(* IEC 61131-3 sources: RL_MAR/experiments/results/ablation/Ablation_antlr_only_deepseek-ai_DeepSeek-V3.2_20260611_164353, 94 files *)

(* ---- hard_92.st ---- *)
FUNCTION_BLOCK FB_BreakerControlSystem
VAR_INPUT
    B10_1_Trip : BOOL;
    B10_1_Close : BOOL;
    B10_2_Trip : BOOL;
    B10_2_Close : BOOL;
    B10_12_Trip : BOOL;
    B10_12_Close : BOOL;
    B54_Trip : BOOL;
    B54_Close : BOOL;
    B55_Trip : BOOL;
    B55_Close : BOOL;
    B56_Trip : BOOL;
    B56_Close : BOOL;
    B57_Trip : BOOL;
    B57_Close : BOOL;
END_VAR

VAR_OUTPUT
    Point_1a : INT;
    Point_2a : INT;
    Point_3a : INT;
    Point_4a : INT;
    B10_1_Opened : BOOL;
    B10_1_Closed : BOOL;
    B10_2_Opened : BOOL;
    B10_2_Closed : BOOL;
    B10_12_Opened : BOOL;
    B10_12_Closed : BOOL;
    B54_Opened : BOOL;
    B54_Closed : BOOL;
    B55_Opened : BOOL;
    B55_Closed : BOOL;
    B56_Opened : BOOL;
    B56_Closed : BOOL;
    B57_Opened : BOOL;
    B57_Closed : BOOL;
END_VAR

VAR
    b10_1_state : BOOL := FALSE;
    b10_2_state : BOOL := FALSE;
    b10_12_state : BOOL := FALSE;
    b54_state : BOOL := FALSE;
    b55_state : BOOL := FALSE;
    b56_state : BOOL := FALSE;
    b57_state : BOOL := FALSE;
END_VAR

(* Breaker B10_1 State Management *)
IF B10_1_Trip THEN
    b10_1_state := FALSE;
ELSIF B10_1_Close THEN
    b10_1_state := TRUE;
END_IF;

B10_1_Closed := b10_1_state;
B10_1_Opened := NOT b10_1_state;

(* Breaker B10_2 State Management *)
IF B10_2_Trip THEN
    b10_2_state := FALSE;
ELSIF B10_2_Close THEN
    b10_2_state := TRUE;
END_IF;

B10_2_Closed := b10_2_state;
B10_2_Opened := NOT b10_2_state;

(* Breaker B10_12 State Management *)
IF B10_12_Trip THEN
    b10_12_state := FALSE;
ELSIF B10_12_Close THEN
    b10_12_state := TRUE;
END_IF;

B10_12_Closed := b10_12_state;
B10_12_Opened := NOT b10_12_state;

(* Breaker B54 State Management *)
IF B54_Trip THEN
    b54_state := FALSE;
ELSIF B54_Close THEN
    b54_state := TRUE;
END_IF;

B54_Closed := b54_state;
B54_Opened := NOT b54_state;

(* Breaker B55 State Management *)
IF B55_Trip THEN
    b55_state := FALSE;
ELSIF B55_Close THEN
    b55_state := TRUE;
END_IF;

B55_Closed := b55_state;
B55_Opened := NOT b55_state;

(* Breaker B56 State Management *)
IF B56_Trip THEN
    b56_state := FALSE;
ELSIF B56_Close THEN
    b56_state := TRUE;
END_IF;

B56_Closed := b56_state;
B56_Opened := NOT b56_state;

(* Breaker B57 State Management *)
IF B57_Trip THEN
    b57_state := FALSE;
ELSIF B57_Close THEN
    b57_state := TRUE;
END_IF;

B57_Closed := b57_state;
B57_Opened := NOT b57_state;

(* Point Calculations *)
(* Point_1a: B54 closed AND ((B10_12 closed AND B10_1 closed) OR B10_2 closed) *)
IF b54_state AND ((b10_12_state AND b10_1_state) OR b10_2_state) THEN
    Point_1a := 0;
ELSE
    Point_1a := 138;
END_IF;

(* Point_2a: B55 closed AND ((B10_12 closed AND B10_1 closed) OR B10_2 closed) *)
IF b55_state AND ((b10_12_state AND b10_1_state) OR b10_2_state) THEN
    Point_2a := 0;
ELSE
    Point_2a := 138;
END_IF;

(* Point_3a: B56 closed AND ((B10_12 closed AND B10_2 closed) OR B10_1 closed) *)
IF b56_state AND ((b10_12_state AND b10_2_state) OR b10_1_state) THEN
    Point_3a := 0;
ELSE
    Point_3a := 138;
END_IF;

(* Point_4a: B57 closed AND ((B10_12 closed AND B10_2 closed) OR B10_1 closed) *)
IF b57_state AND ((b10_12_state AND b10_2_state) OR b10_1_state) THEN
    Point_4a := 0;
ELSE
    Point_4a := 138;
END_IF;

END_FUNCTION_BLOCK;

(* ---- hard_93.st ---- *)
TYPE ST_CircuitBreakerStates :
STRUCT
    Open_CB2_22KV : BOOL;
    Open_CB1_66KV : BOOL;
    Open_CB_TRSF1 : BOOL;
    Open_CB2_66KV : BOOL;
END_STRUCT
END_TYPE

FUNCTION_BLOCK FB_CircuitControl
VAR_INPUT
    Reset_All_CB : BOOL;
    Current_Fault_on_TRSF1 : INT;
    Current_Fault_on_66BUS1 : INT;
END_VAR

VAR_OUTPUT
    Short_Circuit_TRSF1 : BOOL;
    Short_Circuit_66BUS : BOOL;
    Open_CB1_66KV : BOOL;
    Open_CB2_66KV : BOOL;
    Open_CB_TRSF1 : BOOL;
    Open_CB2_22KV : BOOL;
END_VAR

VAR
    Threshold500 : INT := 500;
    Prev_States : ST_CircuitBreakerStates;
    Next_States : ST_CircuitBreakerStates;
    bShortCircuitDetected : BOOL;
END_VAR

(* 1. SHORT CIRCUIT DETECTION (Independent of Reset) *)
Short_Circuit_66BUS := (Current_Fault_on_66BUS1 > Threshold500);
Short_Circuit_TRSF1 := (Current_Fault_on_TRSF1 > Threshold500);

(* 2. RESET OVERRIDE - All breakers to FALSE (Closed) except CB2_66KV *)
IF Reset_All_CB THEN
    Next_States.Open_CB2_22KV := FALSE;
    Next_States.Open_CB1_66KV := FALSE;
    Next_States.Open_CB_TRSF1 := FALSE;
    Next_States.Open_CB2_66KV := TRUE; (* Per specification *)
ELSE
    (* 3. CALCULATE NEXT STATES BASED ON PREVIOUS SCAN CYCLE *)
    (* Initialize with previous state - prevents rapid switching *)
    Next_States := Prev_States;

    (* Combined short circuit flag for logic simplification *)
    bShortCircuitDetected := Short_Circuit_66BUS OR Short_Circuit_TRSF1;

    (* --- FIRST PASS LOGIC (as per specification order) --- *)
    (* Open_CB2_22KV - First Condition *)
    IF (NOT Prev_States.Open_CB2_22KV) AND
       ((Prev_States.Open_CB1_66KV AND Prev_States.Open_CB_TRSF1) OR Short_Circuit_66BUS) THEN
        Next_States.Open_CB2_22KV := TRUE;
    END_IF;

    (* Open_CB1_66KV - First Condition *)
    IF (NOT Next_States.Open_CB2_22KV) AND
       ((Prev_States.Open_CB1_66KV AND Prev_States.Open_CB_TRSF1) OR Short_Circuit_66BUS) THEN
        Next_States.Open_CB1_66KV := TRUE;
    END_IF;

    (* Open_CB_TRSF1 - First Condition *)
    IF (NOT Next_States.Open_CB2_22KV) AND
       ((Next_States.Open_CB1_66KV AND Prev_States.Open_CB_TRSF1) OR Short_Circuit_66BUS) THEN
        Next_States.Open_CB_TRSF1 := TRUE;
    END_IF;

    (* Open_CB2_66KV - Always TRUE per specification *)
    Next_States.Open_CB2_66KV := TRUE;

    (* --- SECOND PASS LOGIC (Updates as per specification) --- *)
    (* Update Open_CB2_22KV again *)
    IF (NOT Prev_States.Open_CB2_22KV) AND
       ((Next_States.Open_CB2_66KV AND Next_States.Open_CB1_66KV AND Next_States.Open_CB_TRSF1) OR Short_Circuit_TRSF1) THEN
        Next_States.Open_CB2_22KV := TRUE;
    END_IF;

    (* Update Open_CB1_66KV again *)
    IF (NOT Next_States.Open_CB2_22KV) AND
       ((Next_States.Open_CB2_66KV AND Prev_States.Open_CB1_66KV AND Next_States.Open_CB_TRSF1) OR Short_Circuit_TRSF1) THEN
        Next_States.Open_CB1_66KV := TRUE;
    END_IF;

    (* Update Open_CB_TRSF1 again *)
    IF (NOT Next_States.Open_CB2_22KV) AND
       ((Next_States.Open_CB2_66KV AND Next_States.Open_CB1_66KV AND Prev_States.Open_CB_TRSF1) OR Short_Circuit_TRSF1) THEN
        Next_States.Open_CB_TRSF1 := TRUE;
    END_IF;

    (* 4. FAILSAFE: If any short circuit is detected, ensure critical breakers open *)
    IF bShortCircuitDetected THEN
        Next_States.Open_CB1_66KV := TRUE;
        Next_States.Open_CB_TRSF1 := TRUE;
        Next_States.Open_CB2_22KV := TRUE;
    END_IF;
END_IF;

(* 5. ASSIGN NEXT STATES TO OUTPUTS *)
Open_CB2_22KV := Next_States.Open_CB2_22KV;
Open_CB1_66KV := Next_States.Open_CB1_66KV;
Open_CB_TRSF1 := Next_States.Open_CB_TRSF1;
Open_CB2_66KV := Next_States.Open_CB2_66KV;

(* 6. STORE CURRENT STATES FOR NEXT SCAN CYCLE *)
Prev_States := Next_States;

END_FUNCTION_BLOCK;

(* ---- hard_94.st ---- *)
FUNCTION_BLOCK FB_AdvancedCircuitBreakerControl
VAR_INPUT
    S_AL1_P_B1 : BOOL;
    S_AL1_P_B2 : BOOL;
    S_AL1_MCB : BOOL;
    MCB_BUSY : BOOL;
    MCB_ERROR : BOOL;
    S_AL1_MCBR : BOOL;
    MCBR_BUSY : BOOL;
    MCBR_ERROR : BOOL;
    S_AL1_P_B3 : BOOL;
    S_AL1_MCB2 : BOOL;
    S_AL1_MCBR2 : BOOL;
END_VAR
VAR_OUTPUT
    E_AL1_B1 : BOOL;
    PUWS_AL1_B1_PLUS : BOOL;
    PUWS_AL1_B1_RIGHT : BOOL;
    PAS_AL1_PLUS : BOOL;
    PAS_AL1_TURN : BOOL;
END_VAR
VAR
    PPAL1 : BOOL := 1;
    PP0 : BOOL := 1;
    PP1 : BOOL := 0;
    PP2 : BOOL := 0;
    PP3 : BOOL := 0;
    PP4 : BOOL := 0;
    MCB : BOOL := 1;
    PP5 : BOOL := 0;
    PP7 : BOOL := 0;
    PPL3 : BOOL := 0;
    PPL4 : BOOL := 0;
    MCBR : BOOL := 1;
    PPL5 : BOOL := 0;
    PPL7 : BOOL := 0;
    STABLE : BOOL := 0;
    MCB_CONTROL : BOOL;
END_VAR

(* State Transition Logic *)
STABLE := 0;
WHILE (STABLE = 0) DO
    STABLE := 1;

    (* Main Path Transitions *)
    IF (PP0 = 1) AND (NOT MCB_CONTROL) AND (PP1 = 0) THEN
        PP0 := 0;
        PP1 := 1;
        STABLE := 0;
    END_IF;

    IF (PP1 = 1) AND S_AL1_P_B1 AND (PP2 = 0) THEN
        PP1 := 0;
        PP2 := 1;
        STABLE := 0;
    END_IF;

    IF (PP2 = 1) AND S_AL1_P_B2 AND (NOT MCB_CONTROL) AND (PP3 = 0) THEN
        PP2 := 0;
        PP3 := 1;
        STABLE := 0;
    END_IF;

    IF (PP3 = 1) AND S_AL1_MCB AND (PP4 = 0) AND (PP1 = 0) THEN
        PP3 := 0;
        PP4 := 1;
        PP1 := 1;
        STABLE := 0;
    END_IF;

    IF (PP4 = 1) AND (MCB = 1) AND MCB_BUSY AND (PP5 = 0) THEN
        PP4 := 0;
        MCB := 0;
        PP5 := 1;
        STABLE := 0;
    END_IF;

    IF (PP5 = 1) AND S_AL1_MCB2 AND (PP7 = 0) AND (MCB = 0) THEN
        PP5 := 0;
        PP7 := 1;
        MCB := 1;
        STABLE := 0;
    END_IF;

    IF (PP7 = 1) AND S_AL1_P_B3 THEN
        PP7 := 0;
        STABLE := 0;
    END_IF;

    (* Alternative Path Transitions *)
    IF (PP2 = 1) AND S_AL1_P_B2 AND MCB_CONTROL AND (PPL3 = 0) AND (PP1 = 0) THEN
        PP2 := 0;
        PPL3 := 1;
        PP1 := 1;
        STABLE := 0;
    END_IF;

    IF (PPL3 = 1) AND S_AL1_MCBR AND (PPL4 = 0) THEN
        PPL3 := 0;
        PPL4 := 1;
        STABLE := 0;
    END_IF;

    IF (PPL4 = 1) AND (MCBR = 1) AND MCBR_BUSY AND (PPL5 = 0) THEN
        PPL4 := 0;
        MCBR := 0;
        PPL5 := 1;
        STABLE := 0;
    END_IF;

    IF (PPL5 = 1) AND S_AL1_MCBR2 AND (PPL7 = 0) AND (MCBR = 0) THEN
        PPL5 := 0;
        PPL7 := 1;
        MCBR := 1;
        STABLE := 0;
    END_IF;

    IF (PPL7 = 1) AND S_AL1_P_B3 THEN
        PPL7 := 0;
        STABLE := 0;
    END_IF;
END_WHILE;

(* Output Control Logic *)
(* E_AL1_B1 - Circuit Activation *)
IF (PP0 = 1) OR (PP1 = 1) THEN
    E_AL1_B1 := 1;
ELSIF (PP2 = 1) OR (PP3 = 1) OR (PPL3 = 1) THEN
    E_AL1_B1 := 0;
ELSE
    E_AL1_B1 := 0;
END_IF;

(* MCB_CONTROL - Main Circuit Breaker Control *)
IF (PP3 = 1) THEN
    MCB_CONTROL := 1;
ELSIF (PP0 = 1) THEN
    MCB_CONTROL := 0;
END_IF;

(* PAS_AL1_PLUS and PAS_AL1_TURN - Process Activation Signals *)
IF (PPL3 = 1) OR (PPL4 = 1) THEN
    PAS_AL1_PLUS := 1;
    PAS_AL1_TURN := 1;
ELSIF (PP0 = 1) OR (PP3 = 1) OR (PP4 = 1) THEN
    PAS_AL1_PLUS := 0;
    PAS_AL1_TURN := 0;
ELSE
    PAS_AL1_PLUS := 0;
    PAS_AL1_TURN := 0;
END_IF;

(* PUWS_AL1_B1_PLUS - Plus Direction Control *)
IF (PPAL1 = 1) OR (PP2 = 1) THEN
    PUWS_AL1_B1_PLUS := 1;
ELSE
    PUWS_AL1_B1_PLUS := 0;
END_IF;

(* PUWS_AL1_B1_RIGHT - Right Direction Control *)
IF (PPAL1 = 1) OR (PP2 = 1) THEN
    PUWS_AL1_B1_RIGHT := 0;
ELSE
    PUWS_AL1_B1_RIGHT := 0;
END_IF;

END_FUNCTION_BLOCK;

(* ---- hf_1.st ---- *)
FUNCTION_BLOCK StackMin
VAR_INPUT
    push : BOOL;
    pop : BOOL;
    reset : BOOL;
END_VAR
VAR_OUTPUT
    error : BOOL;
    status : WORD;
END_VAR
VAR_IN_OUT
    item : INT;
    stack : ARRAY[0..3] OF INT;
END_VAR
VAR
    top : INT := -1; // Tracks the index of the top element; -1 means empty
    i : INT; // Loop counter
    minIndex : INT; // Index of the minimum value found during pop
    minValue : INT; // Minimum value found during pop
END_VAR

// Reset has highest priority
IF reset THEN
    top := -1;
    error := FALSE;
    status := 16#0000;
ELSIF push THEN
    // Check if stack is full
    IF top >= 3 THEN
        error := TRUE;
        status := 16#8A04;
    ELSE
        // Perform push operation
        top := top + 1;
        stack[top] := item;
        error := FALSE;
        status := 16#0000;
    END_IF;
ELSIF pop THEN
    // Check if stack is empty
    IF top < 0 THEN
        error := TRUE;
        status := 16#8A05;
    ELSE
        // Find minimum value and its index
        minIndex := 0;
        minValue := stack[0];

        i := 1;
        WHILE i <= top DO
            IF stack[i] < minValue THEN
                minValue := stack[i];
                minIndex := i;
            END_IF;
            i := i + 1;
        END_WHILE;

        // Return minimum value via item
        item := minValue;

        // Shift elements down to remove the minimum
        i := minIndex;
        WHILE i < top DO
            stack[i] := stack[i + 1];
            i := i + 1;
        END_WHILE;

        // Decrement top
        top := top - 1;

        error := FALSE;
        status := 16#0000;
    END_IF;
ELSE
    // No operation requested
    error := FALSE;
    status := 16#0000;
END_IF;

END_FUNCTION_BLOCK

(* ---- hf_10.st ---- *)
FUNCTION_BLOCK FloatingAverage
VAR_INPUT
    cyclicExecution : BOOL; (* When TRUE, periodic reading is performed, and trigger has no effect *)
    trigger : BOOL; (* External trigger signal, reads value upon each rising edge *)
    value : REAL; (* Newly read data value *)
    windowSize : INT; (* The window size for the moving average, which must be between 1 and 100 *)
    reset : BOOL; (* Reset signal, resets the moving average calculation when TRUE *)
END_VAR
VAR_OUTPUT
    average : REAL; (* The moving average *)
    windowSizeReached : BOOL; (* FALSE: Maximum window width not yet reached, TRUE: Maximum window width has been reached *)
    error : BOOL; (* FALSE: No error occurred, TRUE: An error occurred during the execution of FB *)
    status : WORD; (* Status code *)
END_VAR
VAR
    (* Data buffer and management *)
    dataBuffer : ARRAY[1..100] OF REAL; (* Circular buffer for data values *)
    bufferIndex : INT := 1; (* Current insertion index in the circular buffer *)
    sampleCount : INT := 0; (* Number of valid samples currently in the buffer *)
    sum : REAL := 0.0; (* Running sum of the valid samples in the buffer *)

    (* Edge detection and state tracking *)
    triggerPrev : BOOL := FALSE; (* Previous state of trigger for rising edge detection *)
    cyclicPrev : BOOL := FALSE; (* Previous state of cyclicExecution for edge detection *)

    (* Internal validated window size *)
    internalWindowSize : INT := 1;
END_VAR

(* ================================ *)
(* RESET LOGIC - Highest Priority   *)
(* ================================ *)
IF reset THEN
    (* Clear the data buffer *)
    FOR bufferIndex := 1 TO 100 DO
        dataBuffer[bufferIndex] := 0.0;
    END_FOR;

    (* Reset all internal state variables *)
    bufferIndex := 1;
    sampleCount := 0;
    sum := 0.0;
    triggerPrev := FALSE;
    cyclicPrev := FALSE;

    (* Reset outputs *)
    average := 0.0;
    windowSizeReached := FALSE;
    error := FALSE;
    status := 16#0000; (* Execution successful *)

    (* Validate and set internal window size after reset *)
    IF (windowSize >= 1) AND (windowSize <= 100) THEN
        internalWindowSize := windowSize;
    ELSE
        internalWindowSize := 1; (* Default to minimum valid size *)
    END_IF;

    RETURN; (* Exit function block after reset *)
END_IF;

(* ================================ *)
(* WINDOW SIZE VALIDATION           *)
(* ================================ *)
IF (windowSize < 1) OR (windowSize > 100) THEN
    error := TRUE;
    status := 16#8200; (* Window length setting error *)
    average := 0.0;
    windowSizeReached := FALSE;
    RETURN; (* Exit function block on error *)
ELSE
    error := FALSE;
    status := 16#0000; (* Execution successful *)
    internalWindowSize := windowSize;
END_IF;

(* ================================ *)
(* DATA ACQUISITION LOGIC           *)
(* ================================ *)
IF cyclicExecution THEN
    (* Cyclic mode: process every scan *)
    IF NOT cyclicPrev THEN
        cyclicPrev := TRUE; (* Set for next scan *)

        (* Store the old value that will be overwritten *)
        oldValue : REAL;
        IF sampleCount >= internalWindowSize THEN
            (* Buffer is full, calculate index of oldest value to be overwritten *)
            oldValue := dataBuffer[((bufferIndex - internalWindowSize - 1 + 100) MOD 100) + 1];
        ELSE
            oldValue := 0.0; (* No value to remove when buffer not full *)
        END_IF;

        (* Update buffer with new value *)
        dataBuffer[bufferIndex] := value;

        (* Update running sum *)
        sum := sum + value - oldValue;

        (* Update buffer index (circular) *)
        bufferIndex := (bufferIndex MOD 100) + 1;

        (* Update sample count (capped at window size) *)
        IF sampleCount < internalWindowSize THEN
            sampleCount := sampleCount + 1;
        END_IF;
    END_IF;

    (* Reset trigger edge detection in cyclic mode *)
    triggerPrev := FALSE;
ELSE
    (* Triggered mode: only process on rising edge of trigger *)
    cyclicPrev := FALSE; (* Reset cyclic edge detection *)

    IF trigger AND NOT triggerPrev THEN
        (* Rising edge detected *)
        triggerPrev := TRUE;

        (* Store the old value that will be overwritten *)
        oldValue : REAL;
        IF sampleCount >= internalWindowSize THEN
            (* Buffer is full, calculate index of oldest value to be overwritten *)
            oldValue := dataBuffer[((bufferIndex - internalWindowSize - 1 + 100) MOD 100) + 1];
        ELSE
            oldValue := 0.0; (* No value to remove when buffer not full *)
        END_IF;

        (* Update buffer with new value *)
        dataBuffer[bufferIndex] := value;

        (* Update running sum *)
        sum := sum + value - oldValue;

        (* Update buffer index (circular) *)
        bufferIndex := (bufferIndex MOD 100) + 1;

        (* Update sample count (capped at window size) *)
        IF sampleCount < internalWindowSize THEN
            sampleCount := sampleCount + 1;
        END_IF;
    ELSIF NOT trigger THEN
        (* Reset edge detection when trigger goes low *)
        triggerPrev := FALSE;
    END_IF;
END_IF;

(* ================================ *)
(* AVERAGE CALCULATION              *)
(* ================================ *)
IF sampleCount > 0 THEN
    (* Safe division - sampleCount is guaranteed > 0 *)
    average := sum / INT_TO_REAL(sampleCount);

    (* Update windowSizeReached flag *)
    windowSizeReached := (sampleCount >= internalWindowSize);
ELSE
    (* No samples yet *)
    average := 0.0;
    windowSizeReached := FALSE;
END_IF;

END_FUNCTION_BLOCK;

(* ---- hf_11.st ---- *)
(*
    FUNCTION_BLOCK: FB_BottleProcessing
    PURPOSE: Sequential control for a bottle processing line with five stages.
    STATES: 0=Waiting, 1=Cleaning, 2=Filling, 3=Capping, 4=Packing, 5=Completed.
    AUTHOR: Senior PLC Commissioning Engineer
    STANDARD: IEC 61131-3
*)

FUNCTION_BLOCK FB_BottleProcessing
VAR_INPUT
    bottleSensor : BOOL;             (* Detects presence of a bottle at the start *)
    cleaningConfirmButton : BOOL;    (* Manual confirmation: Cleaning stage complete *)
    fillingConfirmButton : BOOL;     (* Manual confirmation: Filling stage complete *)
    cappingConfirmButton : BOOL;     (* Manual confirmation: Capping stage complete *)
    packingConfirmButton : BOOL;     (* Manual confirmation: Packing stage complete *)
    finishedButton : BOOL;           (* Manual confirmation: Process ready for next bottle *)
END_VAR

VAR_OUTPUT
    Pump_Motor : BOOL;       (* Controls the cleaning pump *)
    Filling_Valve : BOOL;    (* Controls the liquid filling valve *)
    Capping_Machine : BOOL;  (* Controls the capping mechanism *)
    Packing_Machine : BOOL;  (* Controls the packing system *)
    Completion_Light : BOOL; (* Indicates the entire process is complete *)
END_VAR

VAR
    State : INT := 0; (* 0=Waiting, 1=Cleaning, 2=Filling, 3=Capping, 4=Packing, 5=Completed *)
END_VAR

(* Main State Machine Logic *)
CASE State OF
    0: (* STATE: Waiting for a bottle *)
        (* Deactivate all outputs while waiting *)
        Pump_Motor := FALSE;
        Filling_Valve := FALSE;
        Capping_Machine := FALSE;
        Packing_Machine := FALSE;
        Completion_Light := FALSE;

        (* TRANSITION: A bottle is detected, start cleaning *)
        IF bottleSensor THEN
            Pump_Motor := TRUE;
            State := 1;
        END_IF;

    1: (* STATE: Cleaning *)
        (* ACTION: Pump is running. Ensure other outputs are off. *)
        Pump_Motor := TRUE;
        Filling_Valve := FALSE;
        Capping_Machine := FALSE;
        Packing_Machine := FALSE;
        Completion_Light := FALSE;

        (* TRANSITION: Operator confirms cleaning is done *)
        IF cleaningConfirmButton THEN
            Pump_Motor := FALSE;
            Filling_Valve := TRUE;
            State := 2;
        END_IF;

    2: (* STATE: Filling *)
        (* ACTION: Filling valve is open. Ensure other outputs are off. *)
        Pump_Motor := FALSE;
        Filling_Valve := TRUE;
        Capping_Machine := FALSE;
        Packing_Machine := FALSE;
        Completion_Light := FALSE;

        (* TRANSITION: Operator confirms filling is done *)
        IF fillingConfirmButton THEN
            Filling_Valve := FALSE;
            Capping_Machine := TRUE;
            State := 3;
        END_IF;

    3: (* STATE: Capping *)
        (* ACTION: Capping machine is active. Ensure other outputs are off. *)
        Pump_Motor := FALSE;
        Filling_Valve := FALSE;
        Capping_Machine := TRUE;
        Packing_Machine := FALSE;
        Completion_Light := FALSE;

        (* TRANSITION: Operator confirms capping is done *)
        IF cappingConfirmButton THEN
            Capping_Machine := FALSE;
            Packing_Machine := TRUE;
            State := 4;
        END_IF;

    4: (* STATE: Packing *)
        (* ACTION: Packing machine is active. Ensure other outputs are off. *)
        Pump_Motor := FALSE;
        Filling_Valve := FALSE;
        Capping_Machine := FALSE;
        Packing_Machine := TRUE;
        Completion_Light := FALSE;

        (* TRANSITION: Operator confirms packing is done *)
        IF packingConfirmButton THEN
            Packing_Machine := FALSE;
            Completion_Light := TRUE;
            State := 5;
        END_IF;

    5: (* STATE: Completed *)
        (* ACTION: Light is on to signal completion. Ensure process outputs are off. *)
        Pump_Motor := FALSE;
        Filling_Valve := FALSE;
        Capping_Machine := FALSE;
        Packing_Machine := FALSE;
        Completion_Light := TRUE;

        (* TRANSITION: Operator acknowledges completion, reset for next cycle *)
        IF finishedButton THEN
            Completion_Light := FALSE;
            (* All outputs are already FALSE, explicit reset is redundant but clear *)
            State := 0;
        END_IF;
END_CASE;

END_FUNCTION_BLOCK

(* ---- hf_12.st ---- *)
(*
    FUNCTION_BLOCK: MaterialMixing
    Description: Controls a material proportioning process with manual and automatic operation modes.
    Features:
    - Emergency stop (estop) immediately deactivates all outputs.
    - Manual mode: Toggle control for each valve and the mixing motor via pushbuttons.
    - Automatic mode: Executes a sequenced process based on level sensor and process mode.
    - Includes safety interlocks and diagnostic checks as per hazard analysis.
*)

TYPE
    E_AutoStep : (
        Step_Idle := 0,
        Step_ValveA := 1,
        Step_ValveB := 2,
        Step_ProcessBranch := 3,
        Step_MixMotor := 4,
        Step_ValveD := 5
    );
END_TYPE

FUNCTION_BLOCK MaterialMixing
VAR_INPUT
    estop : BOOL; (* Emergency Stop, TRUE = Normal, FALSE = Stop *)
    opeMode : BOOL; (* Operation Mode, FALSE = Manual, TRUE = Automatic *)
    valveAStart : BOOL; (* Valve A Toggle Command *)
    valveBStart : BOOL; (* Valve B Toggle Command *)
    valveCStart : BOOL; (* Valve C Toggle Command *)
    valveDStart : BOOL; (* Valve D Toggle Command *)
    mixMotorStart : BOOL; (* Mixing Motor Toggle Command *)
    autoStart : BOOL; (* Automatic Sequence Start/Stop Toggle *)
    processMode : BOOL; (* Process Mode, FALSE = Simple Mix, TRUE = Add Material C *)
    levelSensor : INT; (* Liquid Level [cm] *)
    mixMotorComplete : BOOL; (* Mixing Motor Completed Cycle *)
END_VAR
VAR_OUTPUT
    valveARun : BOOL; (* Valve A Command *)
    valveBRun : BOOL; (* Valve B Command *)
    valveCRun : BOOL; (* Valve C Command *)
    valveDRun : BOOL; (* Valve D Command *)
    mixMotorRun : BOOL; (* Mixing Motor Command *)
END_VAR
VAR
    (* Edge detection for manual and auto start buttons *)
    rTrig_ValveAStart : R_TRIG;
    rTrig_ValveBStart : R_TRIG;
    rTrig_ValveCStart : R_TRIG;
    rTrig_ValveDStart : R_TRIG;
    rTrig_MixMotorStart : R_TRIG;
    rTrig_AutoStart : R_TRIG;

    (* Automatic sequence control *)
    xAutoActive : BOOL := FALSE;
    eAutoStep : E_AutoStep := E_AutoStep.Step_Idle;

    (* Safety and diagnostic flags *)
    xLevelSensorFault : BOOL := FALSE;
    xMixMotorTimeoutFault : BOOL := FALSE;
    tMixMotorTimer : TON;
    tMixMotorTimeoutTime : TIME := T#30s; (* Example watchdog time *)

    (* Internal state for manual toggle logic *)
    xManualValveA : BOOL := FALSE;
    xManualValveB : BOOL := FALSE;
    xManualValveC : BOOL := FALSE;
    xManualValveD : BOOL := FALSE;
    xManualMixMotor : BOOL := FALSE;
END_VAR

(*----------------------------------------------------------------------------*)
(* 1. PRIMARY SAFETY: EMERGENCY STOP OVERRIDE                                 *)
(*    All final output commands are gated by the estop signal.                *)
(*----------------------------------------------------------------------------*)
IF NOT estop THEN
    valveARun := FALSE;
    valveBRun := FALSE;
    valveCRun := FALSE;
    valveDRun := FALSE;
    mixMotorRun := FALSE;
    xAutoActive := FALSE;
    eAutoStep := E_AutoStep.Step_Idle;
    RETURN; (* Exit function block immediately on estop *)
END_IF;

(*----------------------------------------------------------------------------*)
(* 2. SENSOR DIAGNOSTICS & PLAUSIBILITY CHECKS                                *)
(*    Implements mitigation for "Sensor Failure or Signal Loss" hazard.       *)
(*----------------------------------------------------------------------------*)
xLevelSensorFault := (levelSensor < 0) OR (levelSensor > 110); (* Example range check *)

(*----------------------------------------------------------------------------*)
(* 3. MODE SELECTION: MANUAL OR AUTOMATIC                                     *)
(*----------------------------------------------------------------------------*)
IF NOT opeMode THEN (* MANUAL MODE *)
    (* Deactivate automatic sequence *)
    xAutoActive := FALSE;
    eAutoStep := E_AutoStep.Step_Idle;

    (* Edge detection for manual toggle buttons *)
    rTrig_ValveAStart(CLK := valveAStart);
    rTrig_ValveBStart(CLK := valveBStart);
    rTrig_ValveCStart(CLK := valveCStart);
    rTrig_ValveDStart(CLK := valveDStart);
    rTrig_MixMotorStart(CLK := mixMotorStart);

    (* Toggle logic for manual control *)
    IF rTrig_ValveAStart.Q THEN
        xManualValveA := NOT xManualValveA;
    END_IF;
    IF rTrig_ValveBStart.Q THEN
        xManualValveB := NOT xManualValveB;
    END_IF;
    IF rTrig_ValveCStart.Q THEN
        xManualValveC := NOT xManualValveC;
    END_IF;
    IF rTrig_ValveDStart.Q THEN
        xManualValveD := NOT xManualValveD;
    END_IF;
    IF rTrig_MixMotorStart.Q THEN
        xManualMixMotor := NOT xManualMixMotor;
    END_IF;

    (* Apply manual commands to outputs *)
    valveARun := xManualValveA;
    valveBRun := xManualValveB;
    valveCRun := xManualValveC;
    valveDRun := xManualValveD;
    mixMotorRun := xManualMixMotor;

ELSE (* AUTOMATIC MODE *)
    (*--------------------------------------------------------------------*)
    (* 4. AUTOMATIC SEQUENCE CONTROL                                      *)
    (*    Implements the specified process flow with state machine.       *)
    (*--------------------------------------------------------------------*)
    (* Edge detection for auto start/stop toggle *)
    rTrig_AutoStart(CLK := autoStart);
    IF rTrig_AutoStart.Q THEN
        xAutoActive := NOT xAutoActive;
        IF xAutoActive THEN
            (* Start sequence: Ensure safe initial state *)
            valveDRun := FALSE; (* Interlock: Close outlet before starting *)
            eAutoStep := E_AutoStep.Step_ValveA;
        ELSE
            (* Stop sequence *)
            eAutoStep := E_AutoStep.Step_Idle;
        END_IF;
    END_IF;

    (* Automatic Sequence State Machine *)
    IF xAutoActive AND NOT xLevelSensorFault THEN
        CASE eAutoStep OF
            E_AutoStep.Step_ValveA:
                valveARun := TRUE;
                IF levelSensor >= 50 THEN
                    valveARun := FALSE;
                    eAutoStep := E_AutoStep.Step_ValveB;
                END_IF;

            E_AutoStep.Step_ValveB:
                valveBRun := TRUE;
                IF levelSensor >= 80 THEN
                    valveBRun := FALSE;
                    eAutoStep := E_AutoStep.Step_ProcessBranch;
                END_IF;

            E_AutoStep.Step_ProcessBranch:
                IF NOT processMode THEN
                    (* Simple Mix Path *)
                    mixMotorRun := TRUE;
                    tMixMotorTimer(IN := TRUE, PT := tMixMotorTimeoutTime);
                    IF mixMotorComplete THEN
                        mixMotorRun := FALSE;
                        tMixMotorTimer(IN := FALSE);
                        eAutoStep := E_AutoStep.Step_ValveD;
                    ELSIF tMixMotorTimer.Q THEN
                        (* Watchdog timeout - fault *)
                        mixMotorRun := FALSE;
                        xMixMotorTimeoutFault := TRUE;
                        xAutoActive := FALSE;
                        eAutoStep := E_AutoStep.Step_Idle;
                    END_IF;
                ELSE
                    (* Process with Material C *)
                    valveCRun := TRUE;
                    IF levelSensor >= 100 THEN
                        valveCRun := FALSE;
                        eAutoStep := E_AutoStep.Step_MixMotor;
                    END_IF;
                END_IF;

            E_AutoStep.Step_MixMotor:
                mixMotorRun := TRUE;
                tMixMotorTimer(IN := TRUE, PT := tMixMotorTimeoutTime);
                IF mixMotorComplete THEN
                    mixMotorRun := FALSE;
                    tMixMotorTimer(IN := FALSE);
                    eAutoStep := E_AutoStep.Step_ValveD;
                ELSIF tMixMotorTimer.Q THEN
                    (* Watchdog timeout - fault *)
                    mixMotorRun := FALSE;
                    xMixMotorTimeoutFault := TRUE;
                    xAutoActive := FALSE;
                    eAutoStep := E_AutoStep.Step_Idle;
                END_IF;

            E_AutoStep.Step_ValveD:
                (* Safety Interlock: Ensure all inlet valves are closed before opening outlet *)
                IF NOT valveARun AND NOT valveBRun AND NOT valveCRun THEN
                    valveDRun := TRUE;
                END_IF;
                (* Sequence completes and resets *)
                xAutoActive := FALSE;
                eAutoStep := E_AutoStep.Step_Idle;

        END_CASE;
    ELSE
        (* Auto not active or sensor fault: Deactivate all automatic outputs *)
        valveARun := FALSE;
        valveBRun := FALSE;
        valveCRun := FALSE;
        mixMotorRun := FALSE;
        tMixMotorTimer(IN := FALSE);
        (* Note: valveDRun is not forced FALSE here to allow manual control or completion *)
    END_IF;

    (* In Automatic Mode, manual toggle states are ignored for outputs *)
    xManualValveA := FALSE;
    xManualValveB := FALSE;
    xManualValveC := FALSE;
    xManualValveD := FALSE;
    xManualMixMotor := FALSE;
END_IF; (* End of Mode Selection *)

(*----------------------------------------------------------------------------*)
(* 5. FINAL OUTPUT OVERRIDES & INTERLOCKS                                     *)
(*    Applies final safety and interlocking rules.                            *)
(*----------------------------------------------------------------------------*)
(* Override all outputs if a critical fault is detected *)
IF xLevelSensorFault OR xMixMotorTimeoutFault THEN
    valveARun := FALSE;
    valveBRun := FALSE;
    valveCRun := FALSE;
    mixMotorRun := FALSE;
    (* valveDRun may be left as-is or also forced FALSE depending on safety assessment *)
END_IF;

(* Independent High-Level Overfill Protection (Conceptual) *)
(* This logic represents a software safety layer. For SIL-rated applications,
   this must be implemented in a separate safety PLC or hardwired circuit. *)
IF levelSensor > 105 THEN (* Example high-level trip point *)
    valveARun := FALSE;
    valveBRun := FALSE;
    valveCRun := FALSE;
    mixMotorRun := FALSE;
END_IF;

END_FUNCTION_BLOCK

(* ---- hf_13.st ---- *)
FUNCTION_BLOCK TON
VAR_INPUT
    IN : BOOL;
    PT : DINT;
    CYCLE_TIME : DINT;
END_VAR
VAR_OUTPUT
    Q : BOOL;
    ET : DINT;
END_VAR
VAR
    elapsedTimeInternal : DINT := 0;
    IN_PREV : BOOL := FALSE;
END_VAR

IF IN THEN
    IF NOT IN_PREV THEN
        elapsedTimeInternal := 0;
    END_IF;

    IF elapsedTimeInternal < PT THEN
        elapsedTimeInternal := elapsedTimeInternal + CYCLE_TIME;
        Q := FALSE;
    ELSE
        elapsedTimeInternal := PT;
        Q := TRUE;
    END_IF;

    ET := elapsedTimeInternal;
ELSE
    Q := FALSE;
    ET := 0;
    elapsedTimeInternal := 0;
END_IF;

IN_PREV := IN;
END_FUNCTION_BLOCK

FUNCTION_BLOCK LightsControl
VAR_INPUT
    button1 : BOOL; (* Automatic (TRUE) / Manual (FALSE) Mode Select *)
    button2 : BOOL; (* Manual Control / Green Light Request *)
    button3 : BOOL; (* Manual Control / Red Light Request *)
    CYCLE_TIME : DINT; (* Time elapsed in the current PLC cycle (in ms) *)
END_VAR
VAR_OUTPUT
    greenLight : BOOL; (* Green indicator light state *)
    redLight : BOOL; (* Red indicator light state *)
    yellowLight : BOOL; (* Yellow indicator light state *)
END_VAR
VAR
    (* Timers for control *)
    timerAuto : TON;
    timerGreen : TON;
    timerRed : TON;
    timerYellow : TON;
    currentState : INT := 0;
    autoRunTimer : BOOL;
END_VAR

(* Initialize timer cycle times *)
timerAuto.CYCLE_TIME := CYCLE_TIME;
timerGreen.CYCLE_TIME := CYCLE_TIME;
timerRed.CYCLE_TIME := CYCLE_TIME;
timerYellow.CYCLE_TIME := CYCLE_TIME;

(* Manual Mode (button1 = FALSE) *)
IF NOT button1 THEN
    (* Reset automatic mode state and timer *)
    currentState := 0;
    autoRunTimer := FALSE;
    timerAuto.IN := FALSE;

    (* CRITICAL: Reset all manual timers at start of every PLC cycle *)
    timerGreen.IN := FALSE;
    timerRed.IN := FALSE;
    timerYellow.IN := FALSE;

    (* Execute manual timers with reset state *)
    timerGreen(IN := FALSE, PT := 1000, CYCLE_TIME := CYCLE_TIME);
    timerRed(IN := FALSE, PT := 2000, CYCLE_TIME := CYCLE_TIME);
    timerYellow(IN := FALSE, PT := 1000, CYCLE_TIME := CYCLE_TIME);

    (* Manual mode logic based on button combinations *)
    IF NOT button2 AND NOT button3 THEN
        (* Both FALSE: All lights off *)
        greenLight := FALSE;
        redLight := FALSE;
        yellowLight := FALSE;

    ELSIF button2 AND NOT button3 THEN
        (* button2 TRUE, button3 FALSE *)
        greenLight := TRUE;
        timerRed.IN := TRUE;
        timerRed(IN := TRUE, PT := 2000, CYCLE_TIME := CYCLE_TIME);
        redLight := timerRed.Q; (* Blinks at 0.5Hz *)
        yellowLight := FALSE;

    ELSIF NOT button2 AND button3 THEN
        (* button2 FALSE, button3 TRUE *)
        redLight := TRUE;
        timerYellow.IN := TRUE;
        timerYellow(IN := TRUE, PT := 1000, CYCLE_TIME := CYCLE_TIME);
        yellowLight := NOT timerYellow.Q; (* Blinks at 1Hz *)
        greenLight := FALSE;

    ELSIF button2 AND button3 THEN
        (* Both TRUE *)
        yellowLight := TRUE;
        timerGreen.IN := TRUE;
        timerGreen(IN := TRUE, PT := 1000, CYCLE_TIME := CYCLE_TIME);
        greenLight := NOT timerGreen.Q; (* Blinks at 1Hz *)
        redLight := FALSE;
    END_IF;

(* Automatic Mode (button1 = TRUE) *)
ELSE
    (* CRITICAL: Reset all manual timers when entering automatic mode *)
    timerGreen.IN := FALSE;
    timerRed.IN := FALSE;
    timerYellow.IN := FALSE;

    (* Execute manual timers with reset state *)
    timerGreen(IN := FALSE, PT := 1000, CYCLE_TIME := CYCLE_TIME);
    timerRed(IN := FALSE, PT := 2000, CYCLE_TIME := CYCLE_TIME);
    timerYellow(IN := FALSE, PT := 1000, CYCLE_TIME := CYCLE_TIME);

    (* Automatic mode state machine *)
    autoRunTimer := TRUE;
    timerAuto.IN := autoRunTimer;
    timerAuto(IN := autoRunTimer, PT := 1000, CYCLE_TIME := CYCLE_TIME);

    (* State transition logic *)
    IF timerAuto.Q THEN
        currentState := currentState + 1;
        IF currentState > 2 THEN
            currentState := 0;
        END_IF;
    END_IF;

    (* State output logic *)
    CASE currentState OF
        0: (* State 0: Green light on for 1 second *)
            greenLight := TRUE;
            redLight := FALSE;
            yellowLight := FALSE;

        1: (* State 1: Red light on for 1 second *)
            greenLight := FALSE;
            redLight := TRUE;
            yellowLight := FALSE;

        2: (* State 2: Yellow light on for 1 second *)
            greenLight := FALSE;
            redLight := FALSE;
            yellowLight := TRUE;
    END_CASE;
END_IF;

END_FUNCTION_BLOCK

(* ---- hf_14.st ---- *)
TYPE T_GARAGE_SLOT:
STRUCT
    Occupied : BOOL;
    VehicleNumber : INT;
END_STRUCT
END_TYPE

TYPE T_TRUCK_INFO:
STRUCT
    row : INT;
    col : INT;
    VehicleNumber : INT;
END_STRUCT
END_TYPE

FUNCTION_BLOCK TruckGarage
VAR_INPUT
    enter_flag : BOOL;
    exit_flag : BOOL;
    VehicleNumber_in : INT;
END_VAR
VAR_OUTPUT
    truck : T_TRUCK_INFO;
END_VAR
VAR_IN_OUT
    garage : ARRAY[1..3, 1..5] OF T_GARAGE_SLOT;
END_VAR
VAR
    i : INT;
    j : INT;
    CurrentState : INT := 0;
    NextState : INT := 0;
    EntryFound : BOOL;
    ExitFound : BOOL;
END_VAR

(* State Definitions *)
(* 0: IDLE, 1: ENTRY_PROCESSING, 2: EXIT_PROCESSING *)

(* State Transition *)
CurrentState := NextState;

CASE CurrentState OF
    0: (* IDLE *)
        (* Clear output *)
        truck.row := 0;
        truck.col := 0;
        truck.VehicleNumber := 0;
        EntryFound := FALSE;
        ExitFound := FALSE;

        (* Priority: Entry over Exit if both flags are active *)
        IF enter_flag THEN
            NextState := 1; (* Go to ENTRY_PROCESSING *)
        ELSIF exit_flag THEN
            NextState := 2; (* Go to EXIT_PROCESSING *)
        ELSE
            NextState := 0; (* Stay in IDLE *)
        END_IF;

    1: (* ENTRY_PROCESSING *)
        (* Search from last row to first, last column to first *)
        i := 3;
        WHILE i >= 1 AND NOT EntryFound DO
            j := 5;
            WHILE j >= 1 AND NOT EntryFound DO
                IF NOT garage[i,j].Occupied THEN
                    (* Allocate space *)
                    garage[i,j].Occupied := TRUE;
                    garage[i,j].VehicleNumber := VehicleNumber_in;
                    EntryFound := TRUE;
                END_IF;
                j := j - 1;
            END_WHILE;
            i := i - 1;
        END_WHILE;
        NextState := 0; (* Always return to IDLE *)

    2: (* EXIT_PROCESSING *)
        (* Search from first row to last, first column to last *)
        i := 1;
        WHILE i <= 3 AND NOT ExitFound DO
            j := 1;
            WHILE j <= 5 AND NOT ExitFound DO
                IF garage[i,j].Occupied THEN
                    (* Release space and output info *)
                    truck.row := i;
                    truck.col := j;
                    truck.VehicleNumber := garage[i,j].VehicleNumber;
                    garage[i,j].Occupied := FALSE;
                    garage[i,j].VehicleNumber := 0;
                    ExitFound := TRUE;
                END_IF;
                j := j + 1;
            END_WHILE;
            i := i + 1;
        END_WHILE;
        NextState := 0; (* Always return to IDLE *)

    ELSE
        NextState := 0; (* Fallback to IDLE *)
END_CASE;

END_FUNCTION_BLOCK

(* ---- hf_15.st ---- *)
FUNCTION_BLOCK FB_MergeBytes
VAR_INPUT
    byteArray : ARRAY[1..20] OF DINT; (* Each DINT element holds one byte value (0-255) *)
END_VAR
VAR_OUTPUT
    dwordArray : ARRAY[1..10] OF DINT; (* Each DINT will hold 4 merged bytes *)
    mergeDwordNum : DINT; (* Actual number of successfully merged double words *)
END_VAR
VAR
    iByteIndex : DINT; (* Index for traversing byteArray *)
    iDwordIndex : DINT; (* Index for traversing dwordArray *)
    iByteInGroup : DINT; (* Index within a 4-byte group (0-3) *)
    tempDword : DINT; (* Temporary storage for building the double word *)
    currentByte : DINT; (* Temporary storage for a single byte value *)
END_VAR
VAR CONSTANT
    BYTE_ARRAY_SIZE : DINT := 20;
    DWORD_ARRAY_SIZE : DINT := 10;
    BYTES_PER_DWORD : DINT := 4;
END_VAR

(* Initialize output count *)
mergeDwordNum := 0;

(* Clear the output array to ensure predictable state *)
FOR iDwordIndex := 1 TO DWORD_ARRAY_SIZE DO
    dwordArray[iDwordIndex] := 0;
END_FOR;

(* Main merging loop *)
iByteIndex := 1;
iDwordIndex := 1;

WHILE (iByteIndex + (BYTES_PER_DWORD - 1) <= BYTE_ARRAY_SIZE) AND (iDwordIndex <= DWORD_ARRAY_SIZE) DO
    (* Initialize the temporary double word for this group *)
    tempDword := 0;

    (* Combine 4 consecutive bytes into one double word *)
    FOR iByteInGroup := 0 TO BYTES_PER_DWORD-1 DO
        (* Extract the lowest 8 bits (one byte) from the DINT element *)
        currentByte := byteArray[iByteIndex + iByteInGroup] AND 16#000000FF;

        (* Shift the byte to its correct position and OR it into the temporary double word *)
        tempDword := tempDword OR SHL(currentByte, iByteInGroup * 8);
    END_FOR;

    (* Store the merged double word and update counters *)
    dwordArray[iDwordIndex] := tempDword;
    mergeDwordNum := mergeDwordNum + 1;

    (* Move to the next group of bytes and the next double word slot *)
    iByteIndex := iByteIndex + BYTES_PER_DWORD;
    iDwordIndex := iDwordIndex + 1;
END_WHILE;

END_FUNCTION_BLOCK;

(* ---- hf_16.st ---- *)
TYPE
    ST_LinearSegment : STRUCT
        InputMin : REAL;
        InputMax : REAL;
        OutputMin : REAL;
        OutputMax : REAL;
    END_STRUCT;

    E_StatusCode : (
        STATUS_OK := 16#0000,
        STATUS_OUT_OF_RANGE := 16#8001
    );
END_TYPE

FUNCTION_BLOCK FB_LinearizeValue
VAR_INPUT
    InputValue : REAL;
END_VAR

VAR_OUTPUT
    LinearizedValue : REAL := 0.0;
    Error : BOOL := FALSE;
    Status : WORD := 16#0000;
END_VAR

VAR
    // Internal constants for piecewise linear segments
    Segments : ARRAY[1..3] OF ST_LinearSegment := [
        (InputMin := 1200.0, InputMax := 3600.0, OutputMin := 150.0, OutputMax := 240.0),
        (InputMin := 3600.0, InputMax := 4800.0, OutputMin := 240.0, OutputMax := 560.0),
        (InputMin := 4800.0, InputMax := 7000.0, OutputMin := 560.0, OutputMax := 720.0)
    ];
    i : INT;
    FoundSegment : BOOL;
END_VAR

// Reset status flags
Error := FALSE;
Status := E_StatusCode.STATUS_OK;
LinearizedValue := 0.0;
FoundSegment := FALSE;

// Handle out-of-range conditions
IF InputValue < Segments[1].InputMin THEN
    LinearizedValue := Segments[1].OutputMin;
    Error := TRUE;
    Status := E_StatusCode.STATUS_OUT_OF_RANGE;
ELSIF InputValue > Segments[3].InputMax THEN
    LinearizedValue := Segments[3].OutputMax;
    Error := TRUE;
    Status := E_StatusCode.STATUS_OUT_OF_RANGE;
ELSE
    // Find appropriate segment and perform linear interpolation
    FOR i := 1 TO 3 DO
        IF (InputValue >= Segments[i].InputMin) AND (InputValue <= Segments[i].InputMax) THEN
            LinearizedValue := Segments[i].OutputMin +
                              (InputValue - Segments[i].InputMin) *
                              (Segments[i].OutputMax - Segments[i].OutputMin) /
                              (Segments[i].InputMax - Segments[i].InputMin);
            FoundSegment := TRUE;
            EXIT;
        END_IF;
    END_FOR;

    // If no segment found (should not happen with proper range checking)
    IF NOT FoundSegment THEN
        LinearizedValue := 0.0;
        Error := TRUE;
        Status := E_StatusCode.STATUS_OUT_OF_RANGE;
    END_IF;
END_IF;

END_FUNCTION_BLOCK;

(* ---- hf_17.st ---- *)
TYPE
    E_ErrorCode : WORD := 16#0000;
END_TYPE

FUNCTION_BLOCK FB_WarehouseManagement
VAR_INPUT
    requestIn : BOOL := FALSE;
    requestOut : BOOL := FALSE;
END_VAR

VAR_OUTPUT
    productNum : INT := 0;
    libFreeNum : INT := 9;
    error : BOOL := FALSE;
    status : E_ErrorCode := 16#0000;
END_VAR

VAR_IN_OUT
    library : ARRAY[1..9] OF BOOL;
END_VAR

VAR
    i : INT;
    found : BOOL;
    initDone : BOOL := FALSE;
    errFull : WORD := 16#8001;
    errEmpty : WORD := 16#8002;
END_VAR

(* Initialization - Execute once on first cycle *)
IF NOT initDone THEN
    i := 1;
    WHILE i <= 9 DO
        library[i] := FALSE;
        i := i + 1;
    END_WHILE;
    productNum := 0;
    libFreeNum := 9;
    error := FALSE;
    status := 16#0000;
    initDone := TRUE;
END_IF;

(* Reset error state at start of each cycle *)
error := FALSE;
status := 16#0000;

(* Handle concurrent requests: Input has priority over Output *)
IF requestIn THEN
    (* Storage Full Check *)
    IF productNum >= 9 THEN
        error := TRUE;
        status := errFull;
    ELSE
        (* Search for free position from highest to lowest (9→1) *)
        i := 9;
        found := FALSE;
        WHILE i >= 1 AND NOT found DO
            IF NOT library[i] THEN
                library[i] := TRUE;
                productNum := productNum + 1;
                libFreeNum := libFreeNum - 1;
                found := TRUE;
            END_IF;
            i := i - 1;
        END_WHILE;

        (* Verify search succeeded - safety fallback *)
        IF NOT found THEN
            error := TRUE;
            status := errFull;
        END_IF;
    END_IF;

ELSIF requestOut THEN
    (* Storage Empty Check *)
    IF productNum <= 0 THEN
        error := TRUE;
        status := errEmpty;
    ELSE
        (* Search for occupied position from lowest to highest (1→9) *)
        i := 1;
        found := FALSE;
        WHILE i <= 9 AND NOT found DO
            IF library[i] THEN
                library[i] := FALSE;
                productNum := productNum - 1;
                libFreeNum := libFreeNum + 1;
                found := TRUE;
            END_IF;
            i := i + 1;
        END_WHILE;

        (* Verify search succeeded - safety fallback *)
        IF NOT found THEN
            error := TRUE;
            status := errEmpty;
        END_IF;
    END_IF;
END_IF;

(* Data consistency validation - ensure counters remain synchronized *)
IF libFreeNum + productNum <> 9 THEN
    (* Recovery logic: Recalculate based on actual array state *)
    productNum := 0;
    i := 1;
    WHILE i <= 9 DO
        IF library[i] THEN
            productNum := productNum + 1;
        END_IF;
        i := i + 1;
    END_WHILE;
    libFreeNum := 9 - productNum;
END_IF;

END_FUNCTION_BLOCK;

(* ---- hf_18.st ---- *)
FUNCTION_BLOCK FB_ColorLightControl
{ S7_Optimized_Access := 'TRUE' }
VAR_INPUT
    controlButton : BOOL; // Push button for sequence control
END_VAR

VAR_OUTPUT
    greenLight : BOOL; // Green light control signal
    redLight : BOOL; // Red light control signal
    yellowLight : BOOL; // Yellow light control signal
END_VAR

VAR
    state : INT := 1; // State machine control variable
    lastControlButton : BOOL := FALSE; // Previous button state
END_VAR

// Main logic
// Edge detection for control button
IF controlButton AND NOT lastControlButton THEN
    // State transition logic on rising edge
    CASE state OF
        1: state := 2; // State 1 -> State 2
        2: state := 3; // State 2 -> State 3
        3: state := 4; // State 3 -> State 4
        4: state := 5; // State 4 -> State 5
        5: state := 1; // State 5 -> State 1
    END_CASE;
END_IF;

// Update last button state
lastControlButton := controlButton;

// State execution logic
CASE state OF
    1: // State 1: Green Only
        greenLight := TRUE;
        redLight := FALSE;
        yellowLight := FALSE;
    2: // State 2: Red Only
        greenLight := FALSE;
        redLight := TRUE;
        yellowLight := FALSE;
    3: // State 3: Yellow Only
        greenLight := FALSE;
        redLight := FALSE;
        yellowLight := TRUE;
    4: // State 4: All Lights On
        greenLight := TRUE;
        redLight := TRUE;
        yellowLight := TRUE;
    5: // State 5: All Lights Off
        greenLight := FALSE;
        redLight := FALSE;
        yellowLight := FALSE;
END_CASE;

END_FUNCTION_BLOCK;

(* ---- hf_19.st ---- *)
FUNCTION_BLOCK FB_DatabaseManager
VAR_INPUT
    dataInput : ARRAY[0..5] OF BYTE;
    storeTrigger : BOOL;
    resetTrigger : BOOL;
END_VAR

VAR_OUTPUT
    usedSpace : INT := 0;
    remainingSpace : INT := 20;
    error : BOOL;
    status : WORD;
END_VAR

VAR_IN_OUT
    dataBase : ARRAY[1..20] OF BYTE;
END_VAR

VAR
    dataLength : INT;
    i : INT;
END_VAR

IF resetTrigger THEN
    (* Reset Operation *)
    FOR i := 1 TO 20 DO
        dataBase[i] := 0;
    END_FOR;
    usedSpace := 0;
    remainingSpace := 20;
    error := FALSE;
    status := 0;
ELSIF storeTrigger THEN
    (* Data Storage Operation *)
    dataLength := dataInput[0];

    (* Length Validation *)
    IF (dataLength <= 0) OR (dataLength > 5) THEN
        error := TRUE;
        status := 16#8001;
    ELSE
        (* Space Verification *)
        IF (usedSpace + dataLength) > 20 THEN
            error := TRUE;
            status := 16#8002;
        ELSE
            (* Data Storage *)
            FOR i := 1 TO dataLength DO
                dataBase[usedSpace + i] := dataInput[i];
            END_FOR;

            (* Update Counters and Status *)
            usedSpace := usedSpace + dataLength;
            remainingSpace := 20 - usedSpace;
            error := FALSE;
            status := 0;
        END_IF;
    END_IF;
END_IF;

END_FUNCTION_BLOCK

(* ---- hf_2.st ---- *)
TYPE
    // Define a structure to hold the result of the min/max search
    MinMaxResult : STRUCT
        minValue : DINT;
        minValueIndex : DINT;
        maxValue : DINT;
        maxValueIndex : DINT;
    END_STRUCT;
END_TYPE

FUNCTION_BLOCK FindMinMaxValues
VAR_INPUT
    values : ARRAY[1..10] OF DINT;
END_VAR
VAR_OUTPUT
    minValue : DINT;
    minValueIndex : DINT;
    maxValue : DINT;
    maxValueIndex : DINT;
END_VAR
VAR
    i : INT;
END_VAR

// Initialize with the first element
minValue := values[1];
maxValue := values[1];
minValueIndex := 1;
maxValueIndex := 1;

// Iterate through the remaining elements
FOR i := 2 TO 10 DO
    // Check for new minimum
    IF values[i] < minValue THEN
        minValue := values[i];
        minValueIndex := i;
    END_IF;

    // Check for new maximum
    IF values[i] > maxValue THEN
        maxValue := values[i];
        maxValueIndex := i;
    END_IF;
END_FOR;

END_FUNCTION_BLOCK;

(* ---- hf_20.st ---- *)
FUNCTION_BLOCK FB_ProductionLineControl
VAR_INPUT
    Mode : BOOL; (* FALSE: Manual, TRUE: Automatic *)
    ForwardButton : BOOL; (* Manual forward control button *)
    ReverseButton : BOOL; (* Manual reverse control button *)
    SensorA : BOOL; (* Position sensor at station A *)
    SensorB : BOOL; (* Position sensor at station B *)
    SensorC : BOOL; (* Position sensor at station C *)
    ButtonA : BOOL; (* Process activation button at station A *)
    ButtonB : BOOL; (* Process activation button at station B *)
    ButtonC : BOOL; (* Process activation button at station C *)
END_VAR

VAR_OUTPUT
    MotorForward : BOOL; (* Forward motor control signal *)
    MotorReverse : BOOL; (* Reverse motor control signal *)
    CompletionLight : BOOL; (* Process completion indicator *)
END_VAR

VAR
    State : INT := 0; (* State machine control variable *)
END_VAR

(* Main execution logic *)
CASE State OF
    0: (* Initialization state *)
        MotorForward := FALSE;
        MotorReverse := FALSE;
        CompletionLight := FALSE;
        State := 1;

    1: (* State 1: Manual mode OR Automatic mode waiting at Station A *)
        IF NOT Mode THEN (* Manual Mode *)
            (* Forward motion *)
            IF ForwardButton AND NOT ReverseButton THEN
                MotorForward := TRUE;
                MotorReverse := FALSE;
            (* Reverse motion *)
            ELSIF ReverseButton AND NOT ForwardButton THEN
                MotorForward := FALSE;
                MotorReverse := TRUE;
            (* Stop condition - both buttons pressed or neither pressed *)
            ELSE
                MotorForward := FALSE;
                MotorReverse := FALSE;
            END_IF;
            CompletionLight := FALSE;
        ELSE (* Automatic Mode - State 1: Waiting at Station A *)
            MotorForward := FALSE;
            MotorReverse := FALSE;
            CompletionLight := FALSE;
            IF SensorA THEN
                State := 2; (* Transition to State 2 *)
            END_IF;
        END_IF;

    2: (* State 2: Manual mode OR Automatic mode processing at Station A *)
        IF NOT Mode THEN (* Manual Mode *)
            IF ForwardButton AND NOT ReverseButton THEN
                MotorForward := TRUE;
                MotorReverse := FALSE;
            ELSIF ReverseButton AND NOT ForwardButton THEN
                MotorForward := FALSE;
                MotorReverse := TRUE;
            ELSE
                MotorForward := FALSE;
                MotorReverse := FALSE;
            END_IF;
            CompletionLight := FALSE;
        ELSE (* Automatic Mode - State 2: Processing at Station A *)
            MotorForward := FALSE;
            MotorReverse := FALSE;
            CompletionLight := FALSE;
            IF ButtonA THEN
                MotorForward := TRUE;
                MotorReverse := FALSE;
                State := 3; (* Transition to State 3 *)
            END_IF;
        END_IF;

    3: (* State 3: Manual mode OR Automatic mode moving to Station B *)
        IF NOT Mode THEN (* Manual Mode *)
            IF ForwardButton AND NOT ReverseButton THEN
                MotorForward := TRUE;
                MotorReverse := FALSE;
            ELSIF ReverseButton AND NOT ForwardButton THEN
                MotorForward := FALSE;
                MotorReverse := TRUE;
            ELSE
                MotorForward := FALSE;
                MotorReverse := FALSE;
            END_IF;
            CompletionLight := FALSE;
        ELSE (* Automatic Mode - State 3: Moving to Station B *)
            MotorForward := TRUE;
            MotorReverse := FALSE;
            CompletionLight := FALSE;
            IF SensorB THEN
                MotorForward := FALSE;
                State := 4; (* Transition to State 4 *)
            END_IF;
        END_IF;

    4: (* State 4: Manual mode OR Automatic mode processing at Station B *)
        IF NOT Mode THEN (* Manual Mode *)
            IF ForwardButton AND NOT ReverseButton THEN
                MotorForward := TRUE;
                MotorReverse := FALSE;
            ELSIF ReverseButton AND NOT ForwardButton THEN
                MotorForward := FALSE;
                MotorReverse := TRUE;
            ELSE
                MotorForward := FALSE;
                MotorReverse := FALSE;
            END_IF;
            CompletionLight := FALSE;
        ELSE (* Automatic Mode - State 4: Processing at Station B *)
            MotorForward := FALSE;
            MotorReverse := FALSE;
            CompletionLight := FALSE;
            IF ButtonB THEN
                MotorForward := TRUE;
                MotorReverse := FALSE;
                State := 5; (* Transition to State 5 *)
            END_IF;
        END_IF;

    5: (* State 5: Manual mode OR Automatic mode moving to Station C *)
        IF NOT Mode THEN (* Manual Mode *)
            IF ForwardButton AND NOT ReverseButton THEN
                MotorForward := TRUE;
                MotorReverse := FALSE;
            ELSIF ReverseButton AND NOT ForwardButton THEN
                MotorForward := FALSE;
                MotorReverse := TRUE;
            ELSE
                MotorForward := FALSE;
                MotorReverse := FALSE;
            END_IF;
            CompletionLight := FALSE;
        ELSE (* Automatic Mode - State 5: Moving to Station C *)
            MotorForward := TRUE;
            MotorReverse := FALSE;
            CompletionLight := FALSE;
            IF SensorC THEN
                MotorForward := FALSE;
                State := 6; (* Transition to State 6 *)
            END_IF;
        END_IF;

    6: (* State 6: Manual mode OR Automatic mode processing at Station C *)
        IF NOT Mode THEN (* Manual Mode *)
            IF ForwardButton AND NOT ReverseButton THEN
                MotorForward := TRUE;
                MotorReverse := FALSE;
            ELSIF ReverseButton AND NOT ForwardButton THEN
                MotorForward := FALSE;
                MotorReverse := TRUE;
            ELSE
                MotorForward := FALSE;
                MotorReverse := FALSE;
            END_IF;
            CompletionLight := FALSE;
        ELSE (* Automatic Mode - State 6: Processing at Station C *)
            MotorForward := FALSE;
            MotorReverse := FALSE;
            CompletionLight := FALSE;
            IF ButtonC THEN
                CompletionLight := TRUE;
                State := 7; (* Transition to State 7 *)
            END_IF;
        END_IF;

    7: (* State 7: Manual mode OR Automatic mode cycle completion *)
        IF NOT Mode THEN (* Manual Mode *)
            IF ForwardButton AND NOT ReverseButton THEN
                MotorForward := TRUE;
                MotorReverse := FALSE;
            ELSIF ReverseButton AND NOT ForwardButton THEN
                MotorForward := FALSE;
                MotorReverse := TRUE;
            ELSE
                MotorForward := FALSE;
                MotorReverse := FALSE;
            END_IF;
            CompletionLight := FALSE;
        ELSE (* Automatic Mode - State 7: Cycle Completion *)
            MotorForward := FALSE;
            MotorReverse := FALSE;
            IF NOT SensorC THEN
                CompletionLight := FALSE;
                State := 1; (* Return to State 1 *)
            END_IF;
        END_IF;

END_CASE;

END_FUNCTION_BLOCK

(* ---- hf_21.st ---- *)
(*
FB_SplitNumber
Purpose: Separates a four-digit integer (0-9999) into individual digits and finds the minimum non-zero digit value.
Author: Senior PLC Commissioning Engineer
Date: 2024-06-15
*)

FUNCTION_BLOCK FB_SplitNumber
VAR_INPUT
    InputNumber : INT; (* Input integer value, valid range: 0 to 9999 *)
END_VAR

VAR_OUTPUT
    Thousands : INT; (* Thousands place digit (0-9) *)
    Hundreds : INT;  (* Hundreds place digit (0-9) *)
    Tens : INT;      (* Tens place digit (0-9) *)
    Ones : INT;      (* Ones place digit (0-9) *)
    Min : INT;       (* Minimum non-zero digit among all separated digits *)
    error : BOOL;    (* Error state indicator: TRUE = Input validation failed *)
    status : WORD;   (* Error code: 16#8001 = Input out of range, 16#0000 = No error *)
END_VAR

VAR
    tempNumber : INT; (* Temporary variable for remainder calculations *)
    minValue : INT;   (* Temporary variable for minimum value tracking *)
END_VAR

(* Main execution logic *)
IF (InputNumber < 0) OR (InputNumber > 9999) THEN
    (* Error condition: Input out of valid range *)
    error := TRUE;
    status := 16#8001;

    (* Reset all outputs to zero *)
    Thousands := 0;
    Hundreds := 0;
    Tens := 0;
    Ones := 0;
    Min := 0;
ELSE
    (* Valid input condition *)
    error := FALSE;
    status := 16#0000;

    (* Digit Separation Phase *)
    (* Extract thousands digit using integer division *)
    Thousands := InputNumber / 1000;

    (* Calculate remainder after removing thousands *)
    tempNumber := InputNumber MOD 1000;

    (* Extract hundreds digit *)
    Hundreds := tempNumber / 100;

    (* Calculate remainder after removing hundreds *)
    tempNumber := tempNumber MOD 100;

    (* Extract tens digit *)
    Tens := tempNumber / 10;

    (* Extract ones digit (remainder after removing tens) *)
    Ones := tempNumber MOD 10;

    (* Minimum Non-Zero Digit Detection Phase *)
    (* Initialize with maximum possible INT value *)
    minValue := 32767;

    (* Process thousands digit if non-zero *)
    IF Thousands > 0 THEN
        minValue := minimal(minValue, Thousands);
    END_IF;

    (* Process hundreds digit if non-zero *)
    IF Hundreds > 0 THEN
        minValue := minimal(minValue, Hundreds);
    END_IF;

    (* Process tens digit if non-zero *)
    IF Tens > 0 THEN
        minValue := minimal(minValue, Tens);
    END_IF;

    (* Process ones digit if non-zero *)
    IF Ones > 0 THEN
        minValue := minimal(minValue, Ones);
    END_IF;

    (* Determine final Min output *)
    IF minValue = 32767 THEN
        (* All digits were zero *)
        Min := 0;
    ELSE
        (* Found at least one non-zero digit *)
        Min := minValue;
    END_IF;
END_IF;

END_FUNCTION_BLOCK

(* ---- hf_3.st ---- *)
FUNCTION_BLOCK MultiPumpCtrl
VAR_INPUT
    mode : BOOL;                    // FALSE = Manual, TRUE = Automatic
    start : BOOL;                   // Start button
    stop : BOOL;                    // Stop button (highest priority)
    priorities : ARRAY[1..5] OF INT; // Pump priorities (higher value = higher priority)
    selections : ARRAY[1..5] OF BOOL; // Manual mode selections
END_VAR

VAR_OUTPUT
    RunComds : ARRAY[1..5] OF BOOL; // Pump run commands
END_VAR

VAR
    i : INT;                        // Loop counter
    j : INT;                        // Loop counter for bubble sort
    tempPriority : INT;             // Temporary variable for priority swap
    tempIndex : INT;                // Temporary variable for index swap
    sortedPriorities : ARRAY[1..5] OF INT;  // Copy of priorities for sorting
    sortedIndices : ARRAY[1..5] OF INT;     // Original indices after sorting
END_VAR

// Main logic
IF stop THEN
    // Highest priority: stop all pumps
    FOR i := 1 TO 5 DO
        RunComds[i] := FALSE;
    END_FOR;
ELSIF start THEN
    IF NOT mode THEN
        // Manual mode: directly use selections
        FOR i := 1 TO 5 DO
            RunComds[i] := selections[i];
        END_FOR;
    ELSE
        // Automatic mode: find 3 highest priority pumps

        // Initialize arrays for sorting
        FOR i := 1 TO 5 DO
            sortedPriorities[i] := priorities[i];
            sortedIndices[i] := i;
            RunComds[i] := FALSE;  // Start with all pumps stopped
        END_FOR;

        // Simple bubble sort to sort by priority (descending)
        // This ensures stable selection when priorities are equal
        FOR i := 1 TO 4 DO
            FOR j := i + 1 TO 5 DO
                IF sortedPriorities[j] > sortedPriorities[i] THEN
                    // Swap priorities
                    tempPriority := sortedPriorities[i];
                    sortedPriorities[i] := sortedPriorities[j];
                    sortedPriorities[j] := tempPriority;

                    // Swap corresponding indices
                    tempIndex := sortedIndices[i];
                    sortedIndices[i] := sortedIndices[j];
                    sortedIndices[j] := tempIndex;
                END_IF;
            END_FOR;
        END_FOR;

        // Activate top 3 pumps after sorting
        FOR i := 1 TO 3 DO
            RunComds[sortedIndices[i]] := TRUE;
        END_FOR;
    END_IF;
ELSE
    // start = FALSE: maintain current state (no action)
    // Note: In a real PLC system, you might want to explicitly maintain state
    // but the requirement implies we don't change outputs when start is false
END_IF;

END_FUNCTION_BLOCK;

(* ---- hf_4.st ---- *)
TYPE
    E_Status : WORD
    (
        STATUS_OK := 0,
        STATUS_INVALID_YEAR := 16#8001,
        STATUS_INVALID_MONTH := 16#8002,
        STATUS_INVALID_DAY := 16#8003
    );
END_TYPE

FUNCTION_BLOCK FB_CalculateDayOfYear
VAR_INPUT
    Year : INT;
    Month : INT;
    Day : INT;
END_VAR

VAR_OUTPUT
    DayOfYear : INT;
    error : BOOL;
    status : E_Status;
END_VAR

VAR
    DaysInMonth : ARRAY[1..12] OF INT := [31, 28, 31, 30, 31, 30, 31, 31, 30, 31, 30, 31];
END_VAR

VAR_TEMP
    i : INT;
    bIsLeapYear : BOOL;
    iMaxDayForMonth : INT;
END_VAR

    // Initialize outputs
    DayOfYear := 0;
    error := FALSE;
    status := STATUS_OK;

    // 1. Validate month (highest priority)
    IF (Month < 1) OR (Month > 12) THEN
        error := TRUE;
        status := STATUS_INVALID_MONTH;
        RETURN;
    END_IF;

    // 2. Determine leap year status (needed for day validation)
    // Leap year rule: divisible by 4 AND NOT divisible by 100, OR divisible by 400
    bIsLeapYear := ((Year MOD 4) = 0) AND ((Year MOD 100) <> 0) OR ((Year MOD 400) = 0);

    // 3. Validate day (depends on month and leap year status)
    // Get maximum days for the given month
    iMaxDayForMonth := DaysInMonth[Month];

    // Special handling for February in leap years
    IF (Month = 2) AND bIsLeapYear THEN
        iMaxDayForMonth := 29;
    END_IF;

    // Check day validity: must be positive and not exceed maximum for month
    IF (Day < 1) OR (Day > iMaxDayForMonth) THEN
        error := TRUE;
        status := STATUS_INVALID_DAY;
        RETURN;
    END_IF;

    // 4. Validate year (lowest priority)
    IF (Year < 1000) OR (Year > 3000) THEN
        error := TRUE;
        status := STATUS_INVALID_YEAR;
        RETURN;
    END_IF;

    // 5. Calculate day of year for valid inputs
    // Sum days from all completed months (months before current month)
    FOR i := 1 TO Month-1 DO
        DayOfYear := DayOfYear + DaysInMonth[i];
    END_FOR;

    // Add current day
    DayOfYear := DayOfYear + Day;

    // Add 1 for leap years if date is after February
    IF bIsLeapYear AND (Month > 2) THEN
        DayOfYear := DayOfYear + 1;
    END_IF;

END_FUNCTION_BLOCK

(* ---- hf_5.st ---- *)
FUNCTION_BLOCK SelectSort
VAR_INPUT
    exe : BOOL;
    seq : ARRAY[1..100] OF INT;
END_VAR
VAR_OUTPUT
    error : BOOL;
    status : WORD;
END_VAR
VAR
    i : INT;
    j : INT;
    min_idx : INT;
    temp : INT;
    n : INT := 100;
    seq_local : ARRAY[1..100] OF INT;
    exe_prev : BOOL;
    sortValid : BOOL;
END_VAR

(* Rising edge detection for single execution *)
IF exe AND NOT exe_prev THEN
    (* Initialize outputs to failure state *)
    error := TRUE;
    status := 16#8A01;
    sortValid := TRUE;

    (* Copy input array to local working array *)
    FOR i := 1 TO n DO
        seq_local[i] := seq[i];
    END_FOR;

    (* Selection sort algorithm *)
    FOR i := 1 TO n-1 DO
        min_idx := i;
        FOR j := i+1 TO n DO
            IF seq_local[j] < seq_local[min_idx] THEN
                min_idx := j;
            END_IF;
        END_FOR;

        IF min_idx <> i THEN
            temp := seq_local[i];
            seq_local[i] := seq_local[min_idx];
            seq_local[min_idx] := temp;
        END_IF;
    END_FOR;

    (* Verify array is sorted in ascending order *)
    FOR i := 1 TO n-1 DO
        IF seq_local[i] > seq_local[i+1] THEN
            sortValid := FALSE;
            EXIT;
        END_IF;
    END_FOR;

    (* If verification passed, write back results and set success status *)
    IF sortValid THEN
        FOR i := 1 TO n DO
            seq[i] := seq_local[i];
        END_FOR;

        error := FALSE;
        status := 16#0000;
    END_IF;
END_IF;

(* Update edge detection variable *)
exe_prev := exe;

END_FUNCTION_BLOCK

(* ---- hf_6.st ---- *)
FUNCTION_BLOCK RandomNumberGenerator
VAR_INPUT
    minValue : DINT;
    maxValue : DINT;
    randomSeed_in : DINT;
END_VAR

VAR_OUTPUT
    error : BOOL;
    status : WORD;
    randomNumber : DINT;
END_VAR

VAR
    workingSeed : DINT;
    rangeSize : DINT;
END_VAR

BEGIN
    (* Step 1: Validate input range *)
    IF minValue > maxValue THEN
        error := TRUE;
        status := 16#8200;
        randomNumber := 0;
        RETURN;
    END_IF;

    (* Step 2: Set success status *)
    error := FALSE;
    status := 16#0000;

    (* Step 3: Ensure seed is positive *)
    IF randomSeed_in < 0 THEN
        workingSeed := -randomSeed_in;
    ELSE
        workingSeed := randomSeed_in;
    END_IF;

    (* Step 4: Calculate inclusive range size *)
    rangeSize := maxValue - minValue + 1;

    (* Step 5: Generate pseudo-random value using linear congruential generator *)
    workingSeed := (workingSeed * 1103515245 + 12345) MOD 2147483647;

    (* Step 6: Scale to desired range *)
    randomNumber := minValue + (workingSeed MOD rangeSize);
END_FUNCTION_BLOCK;

(* ---- hf_7.st ---- *)
(* ========================================================================
   FUNCTION_BLOCK: FB_AnalogBatchConverter
   Description: Batch converter for analog input signals with configurable
                scaling and temperature modes. Processes up to 10 channels
                in parallel using configuration arrays.
   Author: Senior PLC Commissioning Engineer
   IEC 61131-3 Compliant
   ======================================================================== *)

FUNCTION_BLOCK FB_AnalogBatchConverter
VAR_INPUT
    (* Number of active channels to process (1..10) *)
    count : INT;
    (* Array of raw analog input values (ADC counts) *)
    analogValues : ARRAY[1..10] OF REAL;
END_VAR

VAR_OUTPUT
    (* Parallel configuration and result arrays *)
    channel_enable : ARRAY[1..10] OF BOOL;
    channel_hiLIM : ARRAY[1..10] OF REAL;
    channel_loLIM : ARRAY[1..10] OF REAL;
    channel_bipolar : ARRAY[1..10] OF BOOL;
    channel_measuringMode : ARRAY[1..10] OF INT;
    channel_retVal : ARRAY[1..10] OF WORD;
    channel_outputValue : ARRAY[1..10] OF REAL;
END_VAR

VAR
    i : INT;                    (* Loop counter *)
    rawValue : REAL;            (* Temporary storage for raw input *)
    normalizedValue : REAL;     (* Normalized value for scaling *)
    rangeInput : REAL;          (* Input range span *)
    rangeOutput : REAL;         (* Output range span *)
    tempOutput : REAL;          (* Temporary output calculation *)
END_VAR

(* Main processing loop *)
FOR i := 1 TO 10 DO
    (* Only process if within active count range AND channel is enabled *)
    IF (i <= count) AND channel_enable[i] THEN
        (* Initialize return value for this channel *)
        channel_retVal[i] := 0;
        rawValue := analogValues[i];

        CASE channel_measuringMode[i] OF
            0: (* Non-temperature measurement *)
                (* Error Check 2: Validate limits *)
                IF channel_hiLIM[i] <= channel_loLIM[i] THEN
                    channel_retVal[i] := 16#8002;  (* Limit violation error *)
                    channel_outputValue[i] := 0.0;  (* Clear output on error *)
                ELSE
                    (* Calculate input range based on bipolar setting *)
                    IF channel_bipolar[i] THEN
                        rangeInput := 55296.0;  (* -27648 to +27648 *)
                        normalizedValue := (rawValue + 27648.0) / rangeInput;
                    ELSE
                        rangeInput := 27648.0;  (* 0 to 27648 *)
                        normalizedValue := rawValue / rangeInput;
                    END_IF;

                    (* Clamp normalized value to valid range [0,1] *)
                    IF normalizedValue < 0.0 THEN
                        normalizedValue := 0.0;
                    ELSIF normalizedValue > 1.0 THEN
                        normalizedValue := 1.0;
                    END_IF;

                    (* Calculate scaled output *)
                    rangeOutput := channel_hiLIM[i] - channel_loLIM[i];
                    channel_outputValue[i] := channel_loLIM[i] + (normalizedValue * rangeOutput);
                END_IF;

            1: (* Standard temperature measurement *)
                channel_outputValue[i] := rawValue / 10.0;

            2: (* Climatic temperature measurement *)
                channel_outputValue[i] := rawValue / 100.0;

            ELSE
                (* Error Check 1: Invalid measuring mode *)
                channel_retVal[i] := 16#8001;  (* Invalid mode error *)
                channel_outputValue[i] := 0.0;  (* Clear output on error *)
        END_CASE;
    ELSE
        (* Channel not enabled or outside active count range *)
        channel_outputValue[i] := 0.0;
        channel_retVal[i] := 0;
    END_IF;
END_FOR;

END_FUNCTION_BLOCK;

(* ---- hf_8.st ---- *)
FUNCTION_BLOCK FB_HexDigitAnalyzer
VAR_INPUT
    InputNumber : INT;
END_VAR
VAR_OUTPUT
    Thousands : INT;
    Hundreds : INT;
    Tens : INT;
    Ones : INT;
    MinDigit : INT;
    error : BOOL;
    status : WORD;
END_VAR
VAR
    tempMin : INT;
    digitVal : INT;
END_VAR

(* Input Validation *)
IF (InputNumber < 0) OR (InputNumber > 9999) THEN
    (* Error Condition *)
    error := TRUE;
    status := 16#8001;
    Thousands := 0;
    Hundreds := 0;
    Tens := 0;
    Ones := 0;
    MinDigit := 0;
ELSE
    (* Valid Input Processing *)
    error := FALSE;
    status := 16#0000;

    (* Digit Separation *)
    Thousands := InputNumber / 1000;
    Hundreds := (InputNumber MOD 1000) / 100;
    Tens := (InputNumber MOD 100) / 10;
    Ones := InputNumber MOD 10;

    (* Minimum Non-Zero Digit Detection *)
    tempMin := 32767; (* Maximum INT value *)

    (* Check Thousands digit *)
    digitVal := Thousands;
    IF digitVal <> 0 THEN
        tempMin := minimal(tempMin, digitVal);
    END_IF;

    (* Check Hundreds digit *)
    digitVal := Hundreds;
    IF digitVal <> 0 THEN
        tempMin := minimal(tempMin, digitVal);
    END_IF;

    (* Check Tens digit *)
    digitVal := Tens;
    IF digitVal <> 0 THEN
        tempMin := minimal(tempMin, digitVal);
    END_IF;

    (* Check Ones digit *)
    digitVal := Ones;
    IF digitVal <> 0 THEN
        tempMin := minimal(tempMin, digitVal);
    END_IF;

    (* Determine final MinDigit output *)
    IF tempMin = 32767 THEN
        (* No non-zero digits found *)
        MinDigit := 0;
    ELSE
        MinDigit := tempMin;
    END_IF;
END_IF;

END_FUNCTION_BLOCK;

(* ---- hf_9.st ---- *)
TYPE
    // Enumeration for sort direction (for internal clarity)
    SortDirectionEnum : (Ascending, Descending);

    // Enumeration for status codes (mapping to required WORD values)
    ShellSortStatusEnum : (Success := 16#0000, SizeTooSmall := 16#8200, SizeTooLarge := 16#8201);
END_TYPE

FUNCTION_BLOCK ShellSortFB
VAR_INPUT
    // Input Variables
    sortDirection : BOOL;  // FALSE = Ascending, TRUE = Descending
    arr : ARRAY[1..1000] OF DINT;  // Fixed-length input array
END_VAR

VAR_OUTPUT
    // Output Variables
    error : BOOL;  // FALSE: No error, TRUE: Error occurred
    status : WORD;  // Status code (16#0000, 16#8200, or 16#8201)
    sorted_arr : ARRAY[1..1000] OF DINT;  // Sorted output array
END_VAR

VAR
    // Algorithm Variables
    gap : DINT;
    i : DINT;
    j : DINT;
    temp : DINT;
    n : DINT := 1000;  // Fixed array size
    dirMultiplier : DINT;  // Direction multiplier for comparison

    // Internal State
    internalStatus : ShellSortStatusEnum;
END_VAR

// 1. Copy input array to output array
sorted_arr := arr;

// 2. Initialize default status (no error)
error := FALSE;
status := 16#0000;
internalStatus := Success;

// 3. Validate array size against fixed constraints
IF n <= 1 THEN
    error := TRUE;
    internalStatus := SizeTooSmall;
ELSIF n > 1000 THEN
    error := TRUE;
    internalStatus := SizeTooLarge;
END_IF;

// 4. Map internal status to output WORD
CASE internalStatus OF
    Success: status := 16#0000;
    SizeTooSmall: status := 16#8200;
    SizeTooLarge: status := 16#8201;
END_CASE;

// 5. If validation failed, return immediately
IF error THEN
    RETURN;
END_IF;

// 6. Set direction multiplier for comparison logic
// For ascending (sortDirection = FALSE): multiplier = 1
// For descending (sortDirection = TRUE): multiplier = -1
IF sortDirection THEN
    dirMultiplier := -1;
ELSE
    dirMultiplier := 1;
END_IF;

// 7. Implement Shell Sort algorithm with optimized gap sequence for 1000 elements
// Using gap sequence: 1000, 500, 250, 125, 62, 31, 15, 7, 3, 1
gap := 1000;
WHILE gap > 0 DO
    i := gap + 1;
    WHILE i <= n DO
        temp := sorted_arr[i];
        j := i;

        // Modified comparison for direction control
        // (sorted_arr[j - gap] - temp) * dirMultiplier > 0
        // This handles both ascending and descending orders
        WHILE (j > gap) AND ((sorted_arr[j - gap] - temp) * dirMultiplier > 0) DO
            sorted_arr[j] := sorted_arr[j - gap];
            j := j - gap;
        END_WHILE;

        sorted_arr[j] := temp;
        i := i + 1;
    END_WHILE;

    // Update gap for next iteration
    CASE gap OF
        1000: gap := 500;
        500: gap := 250;
        250: gap := 125;
        125: gap := 62;
        62: gap := 31;
        31: gap := 15;
        15: gap := 7;
        7: gap := 3;
        3: gap := 1;
        1: gap := 0;
    END_CASE;
END_WHILE;

END_FUNCTION_BLOCK;

(* ---- med_22.st ---- *)
FUNCTION_BLOCK CottonCandyMachine
VAR_INPUT
    SugarLevel : REAL; (* Input for sugar level *)
    SpinningSpeed : INT; (* Input for spinning speed *)
END_VAR
VAR_OUTPUT
    SugarFeeder : BOOL; (* Output to control sugar feeding *)
    MotorSpeed : INT; (* Output to control spinning motor speed *)
END_VAR

(* No internal variables required for this simple combinational logic *)

(* Sugar feeding control: Activate when sugar level is below 10.0 units *)
SugarFeeder := SugarLevel < 10.0;

(* Motor speed control: Set to input speed if positive, otherwise 0 *)
IF SpinningSpeed > 0 THEN
    MotorSpeed := SpinningSpeed;
ELSE
    MotorSpeed := 0;
END_IF;

END_FUNCTION_BLOCK

(* ---- med_23.st ---- *)
(*
    Smart Irrigation System FUNCTION_BLOCK
    Description: Controls a water pump based on soil moisture sensors and weather forecast.
    Inputs:
        SoilMoistureSensor1, SoilMoistureSensor2 : REAL - Soil moisture readings
        WeatherForecast : INT - 0: Sunny, 1: Rainy, 2: Cloudy
    Output:
        WaterPump : BOOL - TRUE to activate pump
    Internal:
        SoilMoistureThreshold : REAL - Moisture level threshold for irrigation
    Logic:
        1. Rain override: If WeatherForecast = 1, pump is always OFF.
        2. Sunny condition: If WeatherForecast = 0 AND (SoilMoistureSensor1 < Threshold OR SoilMoistureSensor2 < Threshold), pump is ON.
        3. All other conditions: Pump is OFF.
*)

FUNCTION_BLOCK SmartIrrigationSystem
VAR_INPUT
    SoilMoistureSensor1 : REAL;
    SoilMoistureSensor2 : REAL;
    WeatherForecast : INT; (* 0: Sunny, 1: Rainy, 2: Cloudy *)
END_VAR

VAR_OUTPUT
    WaterPump : BOOL;
END_VAR

VAR
    SoilMoistureThreshold : REAL := 30.0;
END_VAR

(* Main Control Logic *)
(* Priority 1: Rain override - pump must be OFF if forecast is rainy *)
IF WeatherForecast = 1 THEN
    WaterPump := FALSE;
(* Priority 2: Sunny condition with dry soil - pump ON if needed *)
ELSIF WeatherForecast = 0 THEN
    IF (SoilMoistureSensor1 < SoilMoistureThreshold) OR (SoilMoistureSensor2 < SoilMoistureThreshold) THEN
        WaterPump := TRUE;
    ELSE
        WaterPump := FALSE;
    END_IF;
(* Priority 3: All other conditions (cloudy or invalid forecast) - pump OFF *)
ELSE
    WaterPump := FALSE;
END_IF;

END_FUNCTION_BLOCK;

(* ---- med_24.st ---- *)
FUNCTION_BLOCK AutomaticDoorControl
VAR_INPUT
    ProximitySensor : BOOL;
    ElapsedTime : DINT; (* Time since last door opening in milliseconds *)
END_VAR

VAR_OUTPUT
    DoorOpen : BOOL;
END_VAR

VAR
    DoorOpenDuration : DINT := 5000; (* 5 seconds in milliseconds *)
    tonDoorTimer : TON; (* Standard on-delay timer *)
    bDoorOpeningRequested : BOOL; (* Internal flag for door opening request *)
END_VAR

(* Timer configuration: Runs when door opening is requested *)
tonDoorTimer(
    IN := bDoorOpeningRequested,
    PT := DINT_TO_TIME(DoorOpenDuration)
);

(* Main control logic *)
IF ProximitySensor AND NOT DoorOpen THEN
    (* Request to open door when sensor active and door is closed *)
    DoorOpen := TRUE;
    bDoorOpeningRequested := TRUE;
END_IF;

IF DoorOpen THEN
    (* Door is currently open *)
    IF ProximitySensor THEN
        (* Sensor still active - keep door open and reset timer *)
        bDoorOpeningRequested := TRUE;
    ELSIF NOT bDoorOpeningRequested OR tonDoorTimer.Q THEN
        (* Close door if:
           1. Opening request was cancelled (sensor inactive), OR
           2. Timer has expired (5 seconds elapsed) *)
        DoorOpen := FALSE;
    END_IF;
END_IF;

(* Reset opening request when door closes *)
IF NOT DoorOpen THEN
    bDoorOpeningRequested := FALSE;
END_IF;

END_FUNCTION_BLOCK

(* ---- med_25.st ---- *)
FUNCTION_BLOCK WastewaterControl
VAR_INPUT
    InFlow : REAL;
    OutFlow : REAL;
    pH : REAL;
    TankLvl : REAL;
END_VAR

VAR_OUTPUT
    Pump1 : BOOL;
    Pump2 : BOOL;
    Valve1 : BOOL;
    Valve2 : BOOL;
END_VAR

VAR
    LowInFlow : REAL := 100.0;
    HighOutFlow : REAL := 90.0;
    DesiredPH : REAL := 7.0;
    HighTankLvl : REAL := 80.0;
END_VAR

// Control logic for Pump1: ON when inlet flow is below threshold
Pump1 := InFlow < LowInFlow;

// Control logic for Pump2: ON when outlet flow is above threshold
Pump2 := OutFlow > HighOutFlow;

// Control logic for Valve1: OPEN when pH is below desired level
Valve1 := pH < DesiredPH;

// Control logic for Valve2: OPEN when tank level is above threshold
Valve2 := TankLvl > HighTankLvl;

END_FUNCTION_BLOCK

(* ---- med_26.st ---- *)
FUNCTION_BLOCK BookSorting
VAR_INPUT
    RFID1 : BOOL;
    RFID2 : BOOL;
    RFID3 : BOOL;
END_VAR

VAR_OUTPUT
    Motor : BOOL;
    Bin1 : BOOL;
    Bin2 : BOOL;
    Bin3 : BOOL;
END_VAR

VAR
    (* Internal variable for consolidated detection logic *)
    bAnyRFIDDetected : BOOL;
END_VAR

(* Main Control Logic *)

(* Determine if any RFID reader is active *)
bAnyRFIDDetected := RFID1 OR RFID2 OR RFID3;

(* Control the conveyor motor *)
Motor := bAnyRFIDDetected;

(* Control sorting bins with explicit priority: RFID1 > RFID2 > RFID3 *)
Bin1 := RFID1;
Bin2 := RFID2 AND NOT RFID1;
Bin3 := RFID3 AND NOT RFID1 AND NOT RFID2;

END_FUNCTION_BLOCK

(* ---- med_27.st ---- *)
FUNCTION_BLOCK FlowerArrangingMachine
VAR_INPUT
    FlowerTypeSensor : INT; (* Input for detecting flower type *)
    FlowerColorSensor : INT; (* Input for detecting flower color *)
END_VAR
VAR_OUTPUT
    ArrangingMechanism : INT; (* Output for controlling arranging mechanism *)
    ConveyorBelt : BOOL; (* Output for controlling conveyor belt *)
END_VAR
VAR
    (* No internal variables required for this logic *)
END_VAR

(* Main control logic *)
IF (FlowerTypeSensor = 1) AND (FlowerColorSensor = 1) THEN
    ArrangingMechanism := 1; (* Red type 1 flower *)
ELSIF (FlowerTypeSensor = 1) AND (FlowerColorSensor = 2) THEN
    ArrangingMechanism := 2; (* Blue type 1 flower *)
ELSIF (FlowerTypeSensor = 2) AND (FlowerColorSensor = 1) THEN
    ArrangingMechanism := 3; (* Red type 2 flower *)
ELSIF (FlowerTypeSensor = 2) AND (FlowerColorSensor = 2) THEN
    ArrangingMechanism := 4; (* Blue type 2 flower *)
ELSE
    ArrangingMechanism := 0; (* Any other combination *)
END_IF;

(* Conveyor belt control based on arranging mechanism *)
ConveyorBelt := (ArrangingMechanism <> 0);

END_FUNCTION_BLOCK;

(* ---- med_28.st ---- *)
FUNCTION_BLOCK HomeBrewingSystem
VAR_INPUT
    TemperatureSensor : REAL;     (* Current temperature measurement in °C *)
    WaterFlowSensor : REAL;       (* Current water flow measurement in units *)
    BrewingStartTime : TIME;      (* Absolute time when brewing started *)
    BrewingDuration : TIME;       (* Total duration of the brewing process *)
END_VAR
VAR_OUTPUT
    HeatingElement : BOOL;        (* Control signal for heating element *)
    AgitationMotor : BOOL;        (* Control signal for agitation motor *)
    HopsDispenser : BOOL;         (* Control signal for hops dispenser *)
    FermentationTank : BOOL;      (* Control signal for fermentation tank *)
END_VAR
VAR
    CurrentTime : TIME;           (* Current system time *)
    ElapsedBrewingTime : TIME;    (* Time elapsed since brewing started *)
END_VAR

(* Calculate elapsed time since brewing started *)
CurrentTime := TIME();
ElapsedBrewingTime := CurrentTime - BrewingStartTime;

(* Control heating element based on temperature *)
IF TemperatureSensor < 65.0 THEN
    HeatingElement := TRUE;
ELSE
    HeatingElement := FALSE;
END_IF;

(* Control agitation motor based on water flow *)
IF WaterFlowSensor > 0.5 THEN
    AgitationMotor := TRUE;
ELSE
    AgitationMotor := FALSE;
END_IF;

(* Control hops dispenser - activate after 5 hours of brewing *)
IF ElapsedBrewingTime >= T#5h AND ElapsedBrewingTime <= BrewingDuration THEN
    HopsDispenser := TRUE;
ELSE
    HopsDispenser := FALSE;
END_IF;

(* Control fermentation tank - activate after 48 hours of brewing *)
IF ElapsedBrewingTime >= T#48h AND ElapsedBrewingTime <= BrewingDuration THEN
    FermentationTank := TRUE;
ELSE
    FermentationTank := FALSE;
END_IF;

END_FUNCTION_BLOCK

(* ---- med_29.st ---- *)
(*
    FUNCTION_BLOCK: DocumentFilingSystem
    DESCRIPTION: Controls an automatic document filing system with a conveyor and four storage bins.
    LOGIC:
        - Conveyor motor runs when a document is present AND a valid category (1-4) is selected.
        - Only the storage bin corresponding to the selected category is activated.
        - All outputs are deactivated when no document is present OR an invalid category is selected.
    AUTHOR: Senior PLC Commissioning Engineer
    VERSION: 1.0
    COMPLIANCE: IEC 61131-3
*)

FUNCTION_BLOCK DocumentFilingSystem
VAR_INPUT
    DocumentInlet : BOOL; (* TRUE when a document is detected at the inlet *)
    CategorySelector : INT; (* Selected document category (1-4) *)
END_VAR
VAR_OUTPUT
    ConveyorMotor : BOOL; (* TRUE to run the conveyor motor *)
    StorageBin1 : BOOL; (* TRUE to activate storage bin 1 *)
    StorageBin2 : BOOL; (* TRUE to activate storage bin 2 *)
    StorageBin3 : BOOL; (* TRUE to activate storage bin 3 *)
    StorageBin4 : BOOL; (* TRUE to activate storage bin 4 *)
END_VAR
VAR
    ValidCategory : BOOL; (* Internal flag for category validation *)
END_VAR

    (* Validate the category selector input *)
    ValidCategory := (CategorySelector >= 1) AND (CategorySelector <= 4);

    (* Main control logic: Process document if present and category is valid *)
    IF DocumentInlet AND ValidCategory THEN
        ConveyorMotor := TRUE; (* Run the conveyor *)

        (* Activate only the selected storage bin *)
        CASE CategorySelector OF
            1:
                StorageBin1 := TRUE;
                StorageBin2 := FALSE;
                StorageBin3 := FALSE;
                StorageBin4 := FALSE;
            2:
                StorageBin1 := FALSE;
                StorageBin2 := TRUE;
                StorageBin3 := FALSE;
                StorageBin4 := FALSE;
            3:
                StorageBin1 := FALSE;
                StorageBin2 := FALSE;
                StorageBin3 := TRUE;
                StorageBin4 := FALSE;
            4:
                StorageBin1 := FALSE;
                StorageBin2 := FALSE;
                StorageBin3 := FALSE;
                StorageBin4 := TRUE;
            ELSE
                (* This ELSE case is a safety fallback, though ValidCategory should prevent it *)
                StorageBin1 := FALSE;
                StorageBin2 := FALSE;
                StorageBin3 := FALSE;
                StorageBin4 := FALSE;
        END_CASE;
    ELSE
        (* No document or invalid category: Deactivate all outputs *)
        ConveyorMotor := FALSE;
        StorageBin1 := FALSE;
        StorageBin2 := FALSE;
        StorageBin3 := FALSE;
        StorageBin4 := FALSE;
    END_IF;

END_FUNCTION_BLOCK

(* ---- med_30.st ---- *)
FUNCTION_BLOCK MuseumClimateControl
VAR_INPUT
    HumiditySensor : REAL;
    TemperatureSensor : REAL;
    LightSensor : BOOL;
END_VAR

VAR_OUTPUT
    HVACSystem : BOOL;
    Humidifier : BOOL;
    Dehumidifier : BOOL;
    LightControl : BOOL;
END_VAR

VAR
    TargetHumidity : REAL := 50.0;
    TargetTemperature : REAL := 20.0;
    LightThreshold : BOOL := TRUE;
END_VAR

(* Humidity Control Logic *)
IF HumiditySensor < TargetHumidity THEN
    Humidifier := TRUE;
    Dehumidifier := FALSE;
ELSIF HumiditySensor > TargetHumidity THEN
    Humidifier := FALSE;
    Dehumidifier := TRUE;
ELSE
    Humidifier := FALSE;
    Dehumidifier := FALSE;
END_IF;

(* Temperature Control Logic *)
IF TemperatureSensor <> TargetTemperature THEN
    HVACSystem := TRUE;
ELSE
    HVACSystem := FALSE;
END_IF;

(* Lighting Control Logic *)
IF LightSensor AND LightThreshold THEN
    LightControl := FALSE;
ELSE
    LightControl := TRUE;
END_IF;

END_FUNCTION_BLOCK

(* ---- med_31.st ---- *)
FUNCTION_BLOCK ChargingStationControl
VAR_INPUT
    EVConnected : BOOL;
    EVVoltage : REAL;
    EVCurrent : REAL;
    EVStateOfCharge : REAL;
    ChargingTimer : TIME;
END_VAR

VAR_OUTPUT
    EVCharging : BOOL;
END_VAR

VAR
    VoltageOK : BOOL;
    CurrentOK : BOOL;
    SOCNotFull : BOOL;
    TimerOK : BOOL;
END_VAR

(* Evaluate individual conditions *)
VoltageOK := EVVoltage > 350.0;
CurrentOK := EVCurrent <= 32.0;
SOCNotFull := EVStateOfCharge < 100.0;
TimerOK := ChargingTimer <= T#2h;

(* Control charging output based on all conditions *)
EVCharging := EVConnected AND VoltageOK AND CurrentOK AND SOCNotFull AND TimerOK;

END_FUNCTION_BLOCK

(* ---- med_32.st ---- *)
FUNCTION_BLOCK GreenhouseWateringSystem
VAR_INPUT
    SoilMoistureSensor : REAL; (* Input for soil moisture level (0-100%) *)
END_VAR

VAR_OUTPUT
    SprinklersOn : BOOL; (* Output for controlling sprinklers - on/off *)
END_VAR

VAR
    ResponseDelay : TIME := T#5s; (* Configurable response delay *)
    DelayTimer : TON; (* Timer for response delay *)
    LastMoistureReading : REAL; (* Stores previous moisture reading *)
    State : INT := 0; (* State machine state: 0=IDLE, 1=TRANSITION_TO_ON, 2=TRANSITION_TO_OFF *)
    TargetSprinklerState : BOOL; (* Target state for sprinklers after delay *)
END_VAR

(* Initialize outputs *)
SprinklersOn := FALSE;

(* Main state machine *)
CASE State OF
    0: (* IDLE - Monitoring state *)
        (* Store current reading for potential future use *)
        LastMoistureReading := SoilMoistureSensor;

        (* Check thresholds and initiate transitions if needed *)
        IF SoilMoistureSensor < 30.0 AND NOT SprinklersOn THEN
            (* Start transition to turn sprinklers ON *)
            TargetSprinklerState := TRUE;
            DelayTimer(IN := TRUE, PT := ResponseDelay);
            State := 1;
        ELSIF SoilMoistureSensor > 70.0 AND SprinklersOn THEN
            (* Start transition to turn sprinklers OFF *)
            TargetSprinklerState := FALSE;
            DelayTimer(IN := TRUE, PT := ResponseDelay);
            State := 2;
        ELSE
            (* No transition needed, ensure timer is reset *)
            DelayTimer(IN := FALSE);
        END_IF;

    1: (* TRANSITION_TO_ON - Waiting to turn sprinklers on *)
        (* Sprinklers remain OFF during transition *)
        SprinklersOn := FALSE;

        (* Check if timer has elapsed *)
        IF DelayTimer.Q THEN
            (* Timer elapsed - complete transition *)
            SprinklersOn := TargetSprinklerState; (* = TRUE *)
            DelayTimer(IN := FALSE);
            State := 0;
        ELSIF SoilMoistureSensor >= 30.0 THEN
            (* Moisture rose above threshold during delay - cancel transition *)
            DelayTimer(IN := FALSE);
            State := 0;
        END_IF;

    2: (* TRANSITION_TO_OFF - Waiting to turn sprinklers off *)
        (* Sprinklers remain ON during transition *)
        SprinklersOn := TRUE;

        (* Check if timer has elapsed *)
        IF DelayTimer.Q THEN
            (* Timer elapsed - complete transition *)
            SprinklersOn := TargetSprinklerState; (* = FALSE *)
            DelayTimer(IN := FALSE);
            State := 0;
        ELSIF SoilMoistureSensor <= 70.0 THEN
            (* Moisture dropped below threshold during delay - cancel transition *)
            DelayTimer(IN := FALSE);
            State := 0;
        END_IF;
END_CASE;

END_FUNCTION_BLOCK;

(* ---- med_33.st ---- *)
FUNCTION_BLOCK RoboticArmColorSorting
VAR_INPUT
    ColorSensorRed : BOOL;   (* Input: Red color sensor *)
    ColorSensorGreen : BOOL;  (* Input: Green color sensor *)
    ColorSensorBlue : BOOL;   (* Input: Blue color sensor *)
END_VAR

VAR_OUTPUT
    RoboticArmMove : BOOL := FALSE;     (* Output: Control for robotic arm movement *)
    BinRed : BOOL := FALSE;           (* Output: Activate red bin *)
    BinGreen : BOOL := FALSE;         (* Output: Activate green bin *)
    BinBlue : BOOL := FALSE;          (* Output: Activate blue bin *)
END_VAR

VAR
    (* Internal variable to track which color is currently active *)
    ActiveColor : INT := 0;
END_VAR

(* Arm movement logic: Move if ANY color sensor is active *)
RoboticArmMove := ColorSensorRed OR ColorSensorGreen OR ColorSensorBlue;

(* Determine which color is detected with priority: Red > Green > Blue *)
IF RoboticArmMove THEN
    IF ColorSensorRed THEN
        ActiveColor := 1;      (* Red has highest priority *)
    ELSIF ColorSensorGreen THEN
        ActiveColor := 2;      (* Green has medium priority *)
    ELSIF ColorSensorBlue THEN
        ActiveColor := 3;      (* Blue has lowest priority *)
    ELSE
        ActiveColor := 0;      (* Safety fallback *)
    END_IF;
ELSE
    ActiveColor := 0;          (* No color detected *)
END_IF;

(* Activate exactly one bin based on the detected color *)
CASE ActiveColor OF
    1:  (* Red detected *)
        BinRed := TRUE;
        BinGreen := FALSE;
        BinBlue := FALSE;

    2:  (* Green detected *)
        BinRed := FALSE;
        BinGreen := TRUE;
        BinBlue := FALSE;

    3:  (* Blue detected *)
        BinRed := FALSE;
        BinGreen := FALSE;
        BinBlue := TRUE;

    ELSE  (* No color detected or error state *)
        BinRed := FALSE;
        BinGreen := FALSE;
        BinBlue := FALSE;
END_CASE;

END_FUNCTION_BLOCK
